KUKA KRL program: EPS_2_26115_SA7010_A_20260219035550.src

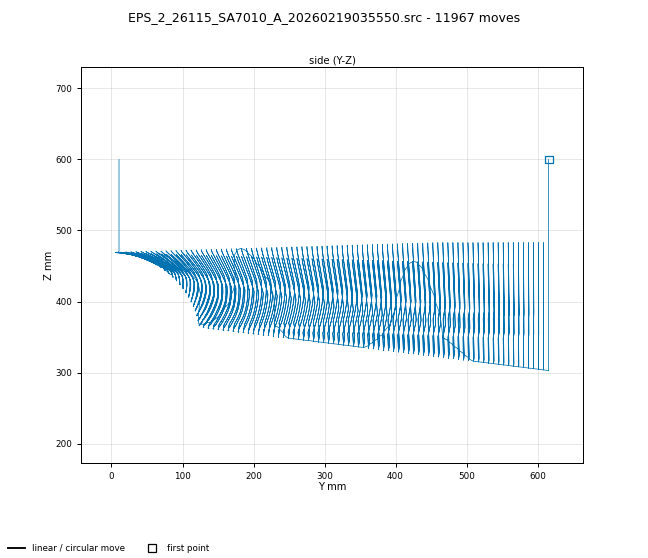
[picture p0: tool path of EPS_2_26115_SA7010_A_20260219035550.src, 11967 of 11969 moves have a stored position in this frame; points joined in program order, loops and branches not executed]
&ACCESS RVP
&REL 4
&COMMENT QRS 19112012
&PARAM EDITMASK = *
DEF PART()
EXT BAS (BAS_COMMAND :IN,REAL :IN )
INT I
BAS (#INITMOV,0 )

;KUKA QRS Post kuka4.cps  Date:22-06-2017 !

File_ID=3066

QRS_PRE_INIT()

;Init var - Until changes are made in qrs_pre_init
Outlet_Square_prg=0
Inlet_1_Square_prg=0
Inlet_2_Square_prg=0
Inlet_3_Square_prg=0
Inlet_4_Square_prg=0
Inlet_5_Square_prg=0

Outlet_1={X 0.000, Y 460.000, Z 382.500, B 0.000, E1 0.000 }
Inlet_1={X 0.000, Y 528.540, Z 352.500, B 0.000, E1 180.000 }
Outlet_1_type=201
Inlet_1_type=201
;QRS#1=Sidecore dimensions
;QRS#2=200-8" PVC SDR 35 Cut Back
;QRS#3=200-8" PVC SDR 35
;QRS#4=
;QRS#5=
;QRS#6=
;QRS#7=
;QRS#8=
;QRS#9=12-08 PSX
;QRS#10=12-08 PSX
;QRS#11=
;QRS#12=
;QRS#13=
;QRS#14=
;QRS#15=
;QRS#16=1220x127x762 2,5'
;QRS#17=EPS Height
;QRS#18=483
;QRS#19=*
;QRS#20= UPDATED VERSION 22-06-2017
;QRS#21=*
Outlet_Square=0100
Inlet_1_Square=0100
Inlet_2_Square=0
Inlet_3_Square=0
Inlet_4_Square=0
Inlet_5_Square=0
Mill_Square=1
Outlet_Square_Prg=214
Inlet_1_Square_prg=204

QRS_INIT()

$ADVANCE=5

; T1
PTP {E1 173.6,E2 173.6}
PTP {X 0,Y 615.497,A -85,B 0,C 180,E1 173.6,E2 173.6,E3 0,E4 0,E5 0,E6 0}
QRS_SPEED_INIT()
LIN {X 0,Y 615.497,Z 600,A -85,B 0,C 180,E1 173.6,E2 173.6,E3 0,E4 0,E5 0,E6 0} C_VEL
LIN {X 0,Y 615.497,Z 312.87,A -85,B 0,C 180,E1 173.6,E2 173.6} C_VEL
LIN {X 0,Y 615.497,Z 304.696,A -85,B 0,C 180,E1 173.6,E2 173.6} C_VEL
LIN {X 0,Y 615.482,Z 302.696,A -85,B 0,C 180,E1 173.414,E2 173.414} C_VEL
LIN {X 0,Y 615.466,Z 302.693,A -85,B 0,C 180,E1 170.801,E2 170.801} C_VEL
LIN {X 0,Y 615.495,Z 302.697,A -85,B 0,C 180,E1 168.139,E2 168.139} C_VEL
LIN {X 0,Y 615.432,Z 302.7,A -85,B 0,C 180,E1 165.449,E2 165.449} C_VEL
LIN {X 0,Y 615.494,Z 302.697,A -85,B 0,C 180,E1 162.73,E2 162.73} C_VEL
LIN {X 0,Y 615.477,Z 302.692,A -85,B 0,C 180,E1 159.967,E2 159.967} C_VEL
LIN {X 0,Y 615.485,Z 302.701,A -85,B 0,C 180,E1 157.651,E2 157.651} C_VEL
LIN {X 0,Y 615.459,Z 302.694,A -85,B 0,C 180,E1 155.007,E2 155.007} C_VEL
LIN {X 0,Y 615.442,Z 302.7,A -85,B 0,C 180,E1 152.083,E2 152.083} C_VEL
LIN {X 0,Y 615.447,Z 302.697,A -85,B 0,C 180,E1 149.838,E2 149.838} C_VEL
LIN {X 0,Y 615.483,Z 302.701,A -85,B 0,C 180,E1 147.542,E2 147.542} C_VEL
LIN {X 0,Y 615.48,Z 302.691,A -85,B 0,C 180,E1 145.184,E2 145.184} C_VEL
LIN {X 0,Y 615.496,Z 302.689,A -85,B 0,C 180,E1 142.758,E2 142.758} C_VEL
LIN {X 0,Y 615.459,Z 302.7,A -85,B 0,C 180,E1 140.247,E2 140.247} C_VEL
LIN {X 0,Y 615.445,Z 302.7,A -85,B 0,C 180,E1 137.643,E2 137.643} C_VEL
LIN {X 0,Y 615.493,Z 302.689,A -85,B 0,C 180,E1 134.932,E2 134.932} C_VEL
LIN {X 0,Y 615.49,Z 302.7,A -85,B 0,C 180,E1 132.08,E2 132.08} C_VEL
LIN {X 0,Y 615.467,Z 302.694,A -85,B 0,C 180,E1 129.75,E2 129.75} C_VEL
LIN {X 0,Y 615.488,Z 302.701,A -85,B 0,C 180,E1 126.936,E2 126.936} C_VEL
LIN {X 0,Y 615.45,Z 302.699,A -85,B 0,C 180,E1 125.617,E2 125.617} C_VEL
LIN {X 0,Y 615.462,Z 303.818,A -85,B 0,C 180,E1 124.697,E2 124.697} C_VEL
LIN {X 0,Y 615.487,Z 307.934,A -85,B 0,C 180,E1 122.33,E2 122.33} C_VEL
LIN {X 0,Y 615.49,Z 313.146,A -85,B 0,C 180,E1 119.405,E2 119.405} C_VEL
LIN {X 0,Y 615.471,Z 317.529,A -85,B 0,C 180,E1 117.041,E2 117.041} C_VEL
LIN {X 0,Y 615.49,Z 322.77,A -85,B 0,C 180,E1 114.271,E2 114.271} C_VEL
LIN {X 0,Y 615.493,Z 328.266,A -85,B 0,C 180,E1 111.431,E2 111.431} C_VEL
LIN {X 0,Y 615.481,Z 333.845,A -85,B 0,C 180,E1 108.602,E2 108.602} C_VEL
LIN {X 0,Y 615.476,Z 339.254,A -85,B 0,C 180,E1 105.905,E2 105.905} C_VEL
LIN {X 0,Y 615.496,Z 344.741,A -85,B 0,C 180,E1 103.2,E2 103.2} C_VEL
LIN {X 0,Y 615.497,Z 348.09,A -85,B 0,C 180,E1 101.568,E2 101.568} C_VEL
LIN {X 0,Y 615.48,Z 362.76,A -85,B 0,C 180,E1 101.234,E2 101.234} C_VEL
LIN {X 0,Y 615.446,Z 375.104,A -85,B 0,C 180,E1 100.825,E2 100.825} C_VEL
LIN {X 0,Y 615.449,Z 387.212,A -85,B 0,C 180,E1 100.278,E2 100.278} C_VEL
LIN {X 0,Y 615.496,Z 398.583,A -85,B 0,C 180,E1 99.613,E2 99.613} C_VEL
LIN {X 0,Y 615.498,Z 408.828,A -85,B 0,C 180,E1 98.867,E2 98.867} C_VEL
LIN {X 0,Y 615.498,Z 418.038,A -85,B 0,C 180,E1 98.04,E2 98.04} C_VEL
LIN {X 0,Y 615.499,Z 426.895,A -85,B 0,C 180,E1 97.057,E2 97.057} C_VEL
LIN {X 0,Y 615.497,Z 434.126,A -85,B 0,C 180,E1 96.062,E2 96.062} C_VEL
LIN {X 0,Y 615.497,Z 438.96,A -85,B 0,C 180,E1 95.241,E2 95.241} C_VEL
LIN {X 0,Y 615.494,Z 443.659,A -85,B 0,C 180,E1 94.256,E2 94.256} C_VEL
LIN {X 0,Y 615.494,Z 447.256,A -85,B 0,C 180,E1 93.273,E2 93.273} C_VEL
LIN {X 0,Y 615.496,Z 449.116,A -85,B 0,C 180,E1 92.617,E2 92.617} C_VEL
LIN {X 0,Y 615.5,Z 450.533,A -85,B 0,C 180,E1 91.963,E2 91.963} C_VEL
LIN {X 0,Y 615.496,Z 452.142,A -85,B 0,C 180,E1 90.654,E2 90.654} C_VEL
LIN {X 0,Y 615.495,Z 452.384,A -85,B 0,C 180,E1 90,E2 90} C_VEL
LIN {X 0,Y 615.495,Z 452.205,A -85,B 0,C 180,E1 89.345,E2 89.345} C_VEL
LIN {X 0,Y 615.5,Z 450.682,A -85,B 0,C 180,E1 88.037,E2 88.037} C_VEL
LIN {X 0,Y 615.498,Z 449.341,A -85,B 0,C 180,E1 87.382,E2 87.382} C_VEL
LIN {X 0,Y 615.496,Z 446.493,A -85,B 0,C 180,E1 86.399,E2 86.399} C_VEL
LIN {X 0,Y 615.498,Z 442.633,A -85,B 0,C 180,E1 85.415,E2 85.415} C_VEL
LIN {X 0,Y 615.498,Z 437.65,A -85,B 0,C 180,E1 84.43,E2 84.43} C_VEL
LIN {X 0,Y 615.496,Z 431.208,A -85,B 0,C 180,E1 83.418,E2 83.418} C_VEL
LIN {X 0,Y 615.497,Z 423.535,A -85,B 0,C 180,E1 82.454,E2 82.454} C_VEL
LIN {X 0,Y 615.498,Z 413.757,A -85,B 0,C 180,E1 81.463,E2 81.463} C_VEL
LIN {X 0,Y 615.498,Z 403.491,A -85,B 0,C 180,E1 80.636,E2 80.636} C_VEL
LIN {X 0,Y 615.459,Z 391.933,A -85,B 0,C 180,E1 79.888,E2 79.888} C_VEL
LIN {X 0,Y 615.436,Z 380.369,A -85,B 0,C 180,E1 79.304,E2 79.304} C_VEL
LIN {X 0,Y 615.462,Z 368.441,A -85,B 0,C 180,E1 78.848,E2 78.848} C_VEL
LIN {X 0,Y 615.491,Z 356.38,A -85,B 0,C 180,E1 78.515,E2 78.515} C_VEL
LIN {X 0,Y 615.497,Z 348.102,A -85,B 0,C 180,E1 78.348,E2 78.348} C_VEL
LIN {X 0,Y 615.474,Z 343.454,A -85,B 0,C 180,E1 76.074,E2 76.074} C_VEL
LIN {X 0,Y 615.463,Z 338.059,A -85,B 0,C 180,E1 73.413,E2 73.413} C_VEL
LIN {X 0,Y 615.49,Z 332.571,A -85,B 0,C 180,E1 70.662,E2 70.662} C_VEL
LIN {X 0,Y 615.473,Z 327.065,A -85,B 0,C 180,E1 67.863,E2 67.863} C_VEL
LIN {X 0,Y 615.488,Z 322.94,A -85,B 0,C 180,E1 65.728,E2 65.728} C_VEL
LIN {X 0,Y 615.474,Z 317.697,A -85,B 0,C 180,E1 62.958,E2 62.958} C_VEL
LIN {X 0,Y 615.492,Z 312.599,A -85,B 0,C 180,E1 60.205,E2 60.205} C_VEL
LIN {X 0,Y 615.488,Z 307.869,A -85,B 0,C 180,E1 57.543,E2 57.543} C_VEL
LIN {X 0,Y 615.467,Z 303.766,A -85,B 0,C 180,E1 55.184,E2 55.184} C_VEL
LIN {X 0,Y 615.454,Z 302.7,A -85,B 0,C 180,E1 54.382,E2 54.382} C_VEL
LIN {X 0,Y 615.449,Z 302.698,A -85,B 0,C 180,E1 51.929,E2 51.929} C_VEL
LIN {X 0,Y 615.49,Z 302.695,A -85,B 0,C 180,E1 49.394,E2 49.394} C_VEL
LIN {X 0,Y 615.489,Z 302.689,A -85,B 0,C 180,E1 46.756,E2 46.756} C_VEL
LIN {X 0,Y 615.458,Z 302.697,A -85,B 0,C 180,E1 43.995,E2 43.995} C_VEL
LIN {X 0,Y 615.481,Z 302.703,A -85,B 0,C 180,E1 41.095,E2 41.095} C_VEL
LIN {X 0,Y 615.474,Z 302.694,A -85,B 0,C 180,E1 38.906,E2 38.906} C_VEL
LIN {X 0,Y 615.464,Z 302.695,A -85,B 0,C 180,E1 36.427,E2 36.427} C_VEL
LIN {X 0,Y 615.483,Z 302.689,A -85,B 0,C 180,E1 33.535,E2 33.535} C_VEL
LIN {X 0,Y 615.495,Z 302.697,A -85,B 0,C 180,E1 30.919,E2 30.919} C_VEL
LIN {X 0,Y 615.439,Z 302.699,A -85,B 0,C 180,E1 28.443,E2 28.443} C_VEL
LIN {X 0,Y 615.498,Z 302.698,A -85,B 0,C 180,E1 25.572,E2 25.572} C_VEL
LIN {X 0,Y 615.463,Z 302.694,A -85,B 0,C 180,E1 22.846,E2 22.846} C_VEL
LIN {X 0,Y 615.491,Z 302.7,A -85,B 0,C 180,E1 20.56,E2 20.56} C_VEL
LIN {X 0,Y 615.473,Z 302.691,A -85,B 0,C 180,E1 17.957,E2 17.957} C_VEL
LIN {X 0,Y 615.478,Z 302.7,A -85,B 0,C 180,E1 15.226,E2 15.226} C_VEL
LIN {X 0,Y 615.439,Z 302.7,A -85,B 0,C 180,E1 12.531,E2 12.531} C_VEL
LIN {X 0,Y 615.497,Z 302.69,A -85,B 0,C 180,E1 9.862,E2 9.862} C_VEL
LIN {X 0,Y 615.476,Z 302.694,A -85,B 0,C 180,E1 7.216,E2 7.216} C_VEL
LIN {X 0,Y 615.468,Z 302.694,A -85,B 0,C 180,E1 4.585,E2 4.585} C_VEL
LIN {X 0,Y 615.499,Z 302.691,A -85,B 0,C 180,E1 1.963,E2 1.963} C_VEL
LIN {X 0,Y 615.438,Z 302.7,A -85,B 0,C 180,E1 -0.654,E2 -0.654} C_VEL
LIN {X 0,Y 615.447,Z 302.696,A -85,B 0,C 180,E1 -2.618,E2 -2.618} C_VEL
LIN {X 0,Y 615.492,Z 302.7,A -85,B 0,C 180,E1 -5.241,E2 -5.241} C_VEL
LIN {X 0,Y 615.488,Z 302.688,A -85,B 0,C 180,E1 -7.876,E2 -7.876} C_VEL
LIN {X 0,Y 615.477,Z 302.699,A -85,B 0,C 180,E1 -10.527,E2 -10.527} C_VEL
LIN {X 0,Y 615.446,Z 302.699,A -85,B 0,C 180,E1 -12.531,E2 -12.531} C_VEL
LIN {X 0,Y 615.469,Z 302.7,A -85,B 0,C 180,E1 -15.227,E2 -15.227} C_VEL
LIN {X 0,Y 615.47,Z 302.692,A -85,B 0,C 180,E1 -17.958,E2 -17.958} C_VEL
LIN {X 0,Y 615.486,Z 302.699,A -85,B 0,C 180,E1 -20.731,E2 -20.731} C_VEL
LIN {X 0,Y 615.489,Z 302.69,A -85,B 0,C 180,E1 -23.556,E2 -23.556} C_VEL
LIN {X 0,Y 615.499,Z 302.7,A -85,B 0,C 180,E1 -25.715,E2 -25.715} C_VEL
LIN {X 0,Y 615.434,Z 302.7,A -85,B 0,C 180,E1 -28.442,E2 -28.442} C_VEL
LIN {X 0,Y 615.495,Z 302.694,A -85,B 0,C 180,E1 -31.088,E2 -31.088} C_VEL
LIN {X 0,Y 615.481,Z 302.696,A -85,B 0,C 180,E1 -34.023,E2 -34.023} C_VEL
LIN {X 0,Y 615.48,Z 302.689,A -85,B 0,C 180,E1 -36.937,E2 -36.937} C_VEL
LIN {X 0,Y 615.46,Z 302.7,A -85,B 0,C 180,E1 -39.752,E2 -39.752} C_VEL
LIN {X 0,Y 615.444,Z 302.7,A -85,B 0,C 180,E1 -42.357,E2 -42.357} C_VEL
LIN {X 0,Y 615.493,Z 302.689,A -85,B 0,C 180,E1 -45.068,E2 -45.068} C_VEL
LIN {X 0,Y 615.49,Z 302.7,A -85,B 0,C 180,E1 -47.92,E2 -47.92} C_VEL
LIN {X 0,Y 615.468,Z 302.694,A -85,B 0,C 180,E1 -50.249,E2 -50.249} C_VEL
LIN {X 0,Y 615.489,Z 302.7,A -85,B 0,C 180,E1 -53.064,E2 -53.064} C_VEL
LIN {X 0,Y 615.468,Z 302.793,A -85,B 0,C 180,E1 -54.584,E2 -54.584} C_VEL
LIN {X 0,Y 615.448,Z 310.011,A -85,B 0,C 180,E1 -57.152,E2 -57.152} C_VEL
LIN {X 0,Y 615.448,Z 317.785,A -85,B 0,C 180,E1 -59.838,E2 -59.838} C_VEL
LIN {X 0,Y 615.496,Z 325.542,A -85,B 0,C 180,E1 -62.455,E2 -62.455} C_VEL
LIN {X 0,Y 615.467,Z 333.312,A -85,B 0,C 180,E1 -65.008,E2 -65.008} C_VEL
LIN {X 0,Y 615.491,Z 341.513,A -85,B 0,C 180,E1 -67.654,E2 -67.654} C_VEL
LIN {X 0,Y 615.484,Z 349.929,A -85,B 0,C 180,E1 -70.315,E2 -70.315} C_VEL
LIN {X 0,Y 615.491,Z 358.782,A -85,B 0,C 180,E1 -73.072,E2 -73.072} C_VEL
LIN {X 0,Y 615.46,Z 367.555,A -85,B 0,C 180,E1 -75.761,E2 -75.761} C_VEL
LIN {X 0,Y 615.497,Z 376.136,A -85,B 0,C 180,E1 -78.369,E2 -78.369} C_VEL
LIN {X 0,Y 615.497,Z 389.818,A -85,B 0,C 180,E1 -78.64,E2 -78.64} C_VEL
LIN {X 0,Y 615.453,Z 402.97,A -85,B 0,C 180,E1 -79.051,E2 -79.051} C_VEL
LIN {X 0,Y 615.442,Z 414.772,A -85,B 0,C 180,E1 -79.555,E2 -79.555} C_VEL
LIN {X 0,Y 615.489,Z 425.386,A -85,B 0,C 180,E1 -80.138,E2 -80.138} C_VEL
LIN {X 0,Y 615.498,Z 436.23,A -85,B 0,C 180,E1 -80.884,E2 -80.884} C_VEL
LIN {X 0,Y 615.497,Z 446.81,A -85,B 0,C 180,E1 -81.794,E2 -81.794} C_VEL
LIN {X 0,Y 615.498,Z 454.605,A -85,B 0,C 180,E1 -82.619,E2 -82.619} C_VEL
LIN {X 0,Y 615.496,Z 462.202,A -85,B 0,C 180,E1 -83.608,E2 -83.608} C_VEL
LIN {X 0,Y 615.498,Z 469.203,A -85,B 0,C 180,E1 -84.759,E2 -84.759} C_VEL
LIN {X 0,Y 615.494,Z 473.85,A -85,B 0,C 180,E1 -85.743,E2 -85.743} C_VEL
LIN {X 0,Y 615.494,Z 477.398,A -85,B 0,C 180,E1 -86.727,E2 -86.727} C_VEL
LIN {X 0,Y 615.497,Z 479.232,A -85,B 0,C 180,E1 -87.382,E2 -87.382} C_VEL
LIN {X 0,Y 615.5,Z 480.607,A -85,B 0,C 180,E1 -88.037,E2 -88.037} C_VEL
LIN {X 0,Y 615.496,Z 482.173,A -85,B 0,C 180,E1 -89.345,E2 -89.345} C_VEL
LIN {X 0,Y 615.494,Z 482.389,A -85,B 0,C 180,E1 -90,E2 -90} C_VEL
LIN {X 0,Y 615.495,Z 481.58,A -85,B 0,C 180,E1 -91.308,E2 -91.308} C_VEL
LIN {X 0,Y 615.5,Z 480.608,A -85,B 0,C 180,E1 -91.963,E2 -91.963} C_VEL
LIN {X 0,Y 615.497,Z 479.234,A -85,B 0,C 180,E1 -92.617,E2 -92.617} C_VEL
LIN {X 0,Y 615.496,Z 476.351,A -85,B 0,C 180,E1 -93.6,E2 -93.6} C_VEL
LIN {X 0,Y 615.498,Z 472.443,A -85,B 0,C 180,E1 -94.584,E2 -94.584} C_VEL
LIN {X 0,Y 615.499,Z 467.407,A -85,B 0,C 180,E1 -95.569,E2 -95.569} C_VEL
LIN {X 0,Y 615.497,Z 460.869,A -85,B 0,C 180,E1 -96.583,E2 -96.583} C_VEL
LIN {X 0,Y 615.497,Z 453.137,A -85,B 0,C 180,E1 -97.545,E2 -97.545} C_VEL
LIN {X 0,Y 615.498,Z 445.05,A -85,B 0,C 180,E1 -98.371,E2 -98.371} C_VEL
LIN {X 0,Y 615.499,Z 435.174,A -85,B 0,C 180,E1 -99.198,E2 -99.198} C_VEL
LIN {X 0,Y 615.479,Z 423.991,A -85,B 0,C 180,E1 -99.945,E2 -99.945} C_VEL
LIN {X 0,Y 615.441,Z 413.04,A -85,B 0,C 180,E1 -100.527,E2 -100.527} C_VEL
LIN {X 0,Y 615.459,Z 400.783,A -85,B 0,C 180,E1 -101.03,E2 -101.03} C_VEL
LIN {X 0,Y 615.499,Z 388.085,A -85,B 0,C 180,E1 -101.401,E2 -101.401} C_VEL
LIN {X 0,Y 615.497,Z 376.138,A -85,B 0,C 180,E1 -101.63,E2 -101.63} C_VEL
LIN {X 0,Y 615.46,Z 367.556,A -85,B 0,C 180,E1 -104.238,E2 -104.238} C_VEL
LIN {X 0,Y 615.491,Z 358.784,A -85,B 0,C 180,E1 -106.928,E2 -106.928} C_VEL
LIN {X 0,Y 615.487,Z 349.931,A -85,B 0,C 180,E1 -109.684,E2 -109.684} C_VEL
LIN {X 0,Y 615.491,Z 341.513,A -85,B 0,C 180,E1 -112.346,E2 -112.346} C_VEL
LIN {X 0,Y 615.467,Z 333.314,A -85,B 0,C 180,E1 -114.992,E2 -114.992} C_VEL
LIN {X 0,Y 615.496,Z 325.544,A -85,B 0,C 180,E1 -117.544,E2 -117.544} C_VEL
LIN {X 0,Y 615.448,Z 317.787,A -85,B 0,C 180,E1 -120.161,E2 -120.161} C_VEL
LIN {X 0,Y 615.448,Z 310.012,A -85,B 0,C 180,E1 -122.847,E2 -122.847} C_VEL
LIN {X 0,Y 615.466,Z 302.699,A -85,B 0,C 180,E1 -125.465,E2 -125.465} C_VEL
LIN {X 0,Y 615.456,Z 302.697,A -85,B 0,C 180,E1 -128.07,E2 -128.07} C_VEL
LIN {X 0,Y 615.486,Z 302.694,A -85,B 0,C 180,E1 -130.605,E2 -130.605} C_VEL
LIN {X 0,Y 615.491,Z 302.69,A -85,B 0,C 180,E1 -133.243,E2 -133.243} C_VEL
LIN {X 0,Y 615.45,Z 302.698,A -85,B 0,C 180,E1 -136.005,E2 -136.005} C_VEL
LIN {X 0,Y 615.456,Z 302.7,A -85,B 0,C 180,E1 -138.523,E2 -138.523} C_VEL
LIN {X 0,Y 615.475,Z 302.693,A -85,B 0,C 180,E1 -141.095,E2 -141.095} C_VEL
LIN {X 0,Y 615.47,Z 302.695,A -85,B 0,C 180,E1 -143.574,E2 -143.574} C_VEL
LIN {X 0,Y 615.481,Z 302.689,A -85,B 0,C 180,E1 -146.465,E2 -146.465} C_VEL
LIN {X 0,Y 615.498,Z 302.698,A -85,B 0,C 180,E1 -149.081,E2 -149.081} C_VEL
LIN {X 0,Y 615.433,Z 302.7,A -85,B 0,C 180,E1 -151.556,E2 -151.556} C_VEL
LIN {X 0,Y 615.494,Z 302.697,A -85,B 0,C 180,E1 -154.427,E2 -154.427} C_VEL
LIN {X 0,Y 615.467,Z 302.694,A -85,B 0,C 180,E1 -157.155,E2 -157.155} C_VEL
LIN {X 0,Y 615.488,Z 302.703,A -85,B 0,C 180,E1 -159.439,E2 -159.439} C_VEL
LIN {X 0,Y 615.469,Z 302.692,A -85,B 0,C 180,E1 -162.042,E2 -162.042} C_VEL
LIN {X 0,Y 615.472,Z 302.7,A -85,B 0,C 180,E1 -164.774,E2 -164.774} C_VEL
LIN {X 0,Y 615.441,Z 302.7,A -85,B 0,C 180,E1 -167.469,E2 -167.469} C_VEL
LIN {X 0,Y 615.497,Z 302.689,A -85,B 0,C 180,E1 -170.138,E2 -170.138} C_VEL
LIN {X 0,Y 615.48,Z 302.694,A -85,B 0,C 180,E1 -172.784,E2 -172.784} C_VEL
LIN {X 0,Y 615.465,Z 302.694,A -85,B 0,C 180,E1 -175.415,E2 -175.415} C_VEL
LIN {X 0,Y 615.499,Z 302.693,A -85,B 0,C 180,E1 -178.037,E2 -178.037} C_VEL
LIN {X 0,Y 615.436,Z 302.7,A -85,B 0,C 180,E1 -180.654,E2 -180.654} C_VEL
LIN {X 0,Y 615.45,Z 302.696,A -85,B 0,C 180,E1 -182.618,E2 -182.618} C_VEL
LIN {X 0,Y 615.49,Z 302.699,A -85,B 0,C 180,E1 -185.241,E2 -185.241} C_VEL
LIN {X 0,Y 615.482,Z 302.696,A -85,B 0,C 180,E1 -186.586,E2 -186.586} C_VEL
LIN {X 0,Y 614.802,Z 302.843,A -85,B 0,C 180,E1 -187.132,E2 -187.132} C_VEL
LIN {X 0,Y 611.956,Z 303.255,A -85,B 0,C 180,E1 -188.018,E2 -188.018} C_VEL
LIN {X 0,Y 609.562,Z 303.564,A -85,B 0,C 180,E1 -188.73,E2 -188.73} C_VEL
LIN {X 0,Y 608.533,Z 303.681,A -85,B 0,C 180,E1 -189.28,E2 -189.28} C_VEL
LIN {X 0,Y 608.449,Z 303.691,A -85,B 0,C 180,E1 -189.466,E2 -189.466} C_VEL
LIN {X 0,Y 608.458,Z 303.698,A -85,B 0,C 180,E1 -192,E2 -192} C_VEL
LIN {X 0,Y 608.405,Z 303.696,A -85,B 0,C 180,E1 -194.722,E2 -194.722} C_VEL
LIN {X 0,Y 608.452,Z 303.693,A -85,B 0,C 180,E1 -197.477,E2 -197.477} C_VEL
LIN {X 0,Y 608.459,Z 303.693,A -85,B 0,C 180,E1 -200.274,E2 -200.274} C_VEL
LIN {X 0,Y 608.448,Z 303.696,A -85,B 0,C 180,E1 -202.477,E2 -202.477} C_VEL
LIN {X 0,Y 608.434,Z 303.693,A -85,B 0,C 180,E1 -204.572,E2 -204.572} C_VEL
LIN {X 0,Y 608.461,Z 303.694,A -85,B 0,C 180,E1 -207.207,E2 -207.207} C_VEL
LIN {X 0,Y 608.42,Z 303.694,A -85,B 0,C 180,E1 -209.966,E2 -209.966} C_VEL
LIN {X 0,Y 608.457,Z 303.697,A -85,B 0,C 180,E1 -212.524,E2 -212.524} C_VEL
LIN {X 0,Y 608.439,Z 303.692,A -85,B 0,C 180,E1 -215.278,E2 -215.278} C_VEL
LIN {X 0,Y 608.46,Z 303.697,A -85,B 0,C 180,E1 -217.747,E2 -217.747} C_VEL
LIN {X 0,Y 608.425,Z 303.694,A -85,B 0,C 180,E1 -220.328,E2 -220.328} C_VEL
LIN {X 0,Y 608.463,Z 303.69,A -85,B 0,C 180,E1 -223.31,E2 -223.31} C_VEL
LIN {X 0,Y 608.462,Z 303.695,A -85,B 0,C 180,E1 -226.131,E2 -226.131} C_VEL
LIN {X 0,Y 608.455,Z 303.69,A -85,B 0,C 180,E1 -228.825,E2 -228.825} C_VEL
LIN {X 0,Y 608.463,Z 303.697,A -85,B 0,C 180,E1 -231.413,E2 -231.413} C_VEL
LIN {X 0,Y 608.427,Z 303.693,A -85,B 0,C 180,E1 -233.957,E2 -233.957} C_VEL
LIN {X 0,Y 608.389,Z 303.802,A -85,B 0,C 180,E1 -234.72,E2 -234.72} C_VEL
LIN {X 0,Y 608.462,Z 307.941,A -85,B 0,C 180,E1 -237.122,E2 -237.122} C_VEL
LIN {X 0,Y 608.452,Z 313.03,A -85,B 0,C 180,E1 -240.031,E2 -240.031} C_VEL
LIN {X 0,Y 608.43,Z 318.103,A -85,B 0,C 180,E1 -242.802,E2 -242.802} C_VEL
LIN {X 0,Y 608.421,Z 323.038,A -85,B 0,C 180,E1 -245.428,E2 -245.428} C_VEL
LIN {X 0,Y 608.446,Z 328.567,A -85,B 0,C 180,E1 -248.308,E2 -248.308} C_VEL
LIN {X 0,Y 608.422,Z 334.429,A -85,B 0,C 180,E1 -251.298,E2 -251.298} C_VEL
LIN {X 0,Y 608.431,Z 339.626,A -85,B 0,C 180,E1 -253.906,E2 -253.906} C_VEL
LIN {X 0,Y 608.435,Z 345.156,A -85,B 0,C 180,E1 -256.643,E2 -256.643} C_VEL
LIN {X 0,Y 608.449,Z 348.525,A -85,B 0,C 180,E1 -258.296,E2 -258.296} C_VEL
LIN {X 0,Y 608.529,Z 364.411,A -85,B 0,C 180,E1 -258.678,E2 -258.678} C_VEL
LIN {X 0,Y 608.478,Z 376.8,A -85,B 0,C 180,E1 -259.112,E2 -259.112} C_VEL
LIN {X 0,Y 608.454,Z 388.944,A -85,B 0,C 180,E1 -259.687,E2 -259.687} C_VEL
LIN {X 0,Y 608.497,Z 400.074,A -85,B 0,C 180,E1 -260.36,E2 -260.36} C_VEL
LIN {X 0,Y 608.474,Z 409.09,A -85,B 0,C 180,E1 -261.03,E2 -261.03} C_VEL
LIN {X 0,Y 608.464,Z 418.354,A -85,B 0,C 180,E1 -261.866,E2 -261.866} C_VEL
LIN {X 0,Y 608.466,Z 427.327,A -85,B 0,C 180,E1 -262.868,E2 -262.868} C_VEL
LIN {X 0,Y 608.444,Z 434.558,A -85,B 0,C 180,E1 -263.867,E2 -263.867} C_VEL
LIN {X 0,Y 608.462,Z 439.436,A -85,B 0,C 180,E1 -264.699,E2 -264.699} C_VEL
LIN {X 0,Y 608.439,Z 444.18,A -85,B 0,C 180,E1 -265.695,E2 -265.695} C_VEL
LIN {X 0,Y 608.425,Z 447.813,A -85,B 0,C 180,E1 -266.689,E2 -266.689} C_VEL
LIN {X 0,Y 608.425,Z 449.692,A -85,B 0,C 180,E1 -267.352,E2 -267.352} C_VEL
LIN {X 0,Y 608.445,Z 451.127,A -85,B 0,C 180,E1 -268.015,E2 -268.015} C_VEL
LIN {X 0,Y 608.439,Z 452.752,A -85,B 0,C 180,E1 -269.338,E2 -269.338} C_VEL
LIN {X 0,Y 608.435,Z 452.995,A -85,B 0,C 180,E1 -270,E2 -270} C_VEL
LIN {X 0,Y 608.438,Z 452.815,A -85,B 0,C 180,E1 -270.662,E2 -270.662} C_VEL
LIN {X 0,Y 608.445,Z 451.276,A -85,B 0,C 180,E1 -271.986,E2 -271.986} C_VEL
LIN {X 0,Y 608.426,Z 449.918,A -85,B 0,C 180,E1 -272.649,E2 -272.649} C_VEL
LIN {X 0,Y 608.449,Z 447.041,A -85,B 0,C 180,E1 -273.643,E2 -273.643} C_VEL
LIN {X 0,Y 608.433,Z 443.142,A -85,B 0,C 180,E1 -274.638,E2 -274.638} C_VEL
LIN {X 0,Y 608.45,Z 438.111,A -85,B 0,C 180,E1 -275.635,E2 -275.635} C_VEL
LIN {X 0,Y 608.441,Z 431.794,A -85,B 0,C 180,E1 -276.633,E2 -276.633} C_VEL
LIN {X 0,Y 608.475,Z 423.877,A -85,B 0,C 180,E1 -277.633,E2 -277.633} C_VEL
LIN {X 0,Y 608.472,Z 414.035,A -85,B 0,C 180,E1 -278.636,E2 -278.636} C_VEL
LIN {X 0,Y 608.481,Z 403.712,A -85,B 0,C 180,E1 -279.473,E2 -279.473} C_VEL
LIN {X 0,Y 608.471,Z 392.098,A -85,B 0,C 180,E1 -280.229,E2 -280.229} C_VEL
LIN {X 0,Y 608.463,Z 380.492,A -85,B 0,C 180,E1 -280.82,E2 -280.82} C_VEL
LIN {X 0,Y 608.492,Z 368.423,A -85,B 0,C 180,E1 -281.286,E2 -281.286} C_VEL
LIN {X 0,Y 608.537,Z 355.557,A -85,B 0,C 180,E1 -281.639,E2 -281.639} C_VEL
LIN {X 0,Y 608.441,Z 348.536,A -85,B 0,C 180,E1 -281.789,E2 -281.789} C_VEL
LIN {X 0,Y 608.427,Z 343.954,A -85,B 0,C 180,E1 -284.038,E2 -284.038} C_VEL
LIN {X 0,Y 608.405,Z 338.422,A -85,B 0,C 180,E1 -286.785,E2 -286.785} C_VEL
LIN {X 0,Y 608.43,Z 332.89,A -85,B 0,C 180,E1 -289.571,E2 -289.571} C_VEL
LIN {X 0,Y 608.435,Z 327.357,A -85,B 0,C 180,E1 -292.407,E2 -292.407} C_VEL
LIN {X 0,Y 608.421,Z 323.208,A -85,B 0,C 180,E1 -294.572,E2 -294.572} C_VEL
LIN {X 0,Y 608.432,Z 318.269,A -85,B 0,C 180,E1 -297.198,E2 -297.198} C_VEL
LIN {X 0,Y 608.453,Z 313.188,A -85,B 0,C 180,E1 -299.969,E2 -299.969} C_VEL
LIN {X 0,Y 608.46,Z 308.059,A -85,B 0,C 180,E1 -302.879,E2 -302.879} C_VEL
LIN {X 0,Y 608.392,Z 303.954,A -85,B 0,C 180,E1 -305.281,E2 -305.281} C_VEL
LIN {X 0,Y 608.479,Z 303.692,A -85,B 0,C 180,E1 -307.159,E2 -307.159} C_VEL
LIN {X 0,Y 608.446,Z 303.698,A -85,B 0,C 180,E1 -310.328,E2 -310.328} C_VEL
LIN {X 0,Y 608.455,Z 303.69,A -85,B 0,C 180,E1 -312.959,E2 -312.959} C_VEL
LIN {X 0,Y 608.441,Z 303.696,A -85,B 0,C 180,E1 -315.737,E2 -315.737} C_VEL
LIN {X 0,Y 608.417,Z 303.695,A -85,B 0,C 180,E1 -317.935,E2 -317.935} C_VEL
LIN {X 0,Y 608.439,Z 303.699,A -85,B 0,C 180,E1 -320.705,E2 -320.705} C_VEL
LIN {X 0,Y 608.448,Z 303.691,A -85,B 0,C 180,E1 -323.084,E2 -323.084} C_VEL
LIN {X 0,Y 608.464,Z 303.693,A -85,B 0,C 180,E1 -325.53,E2 -325.53} C_VEL
LIN {X 0,Y 608.461,Z 303.691,A -85,B 0,C 180,E1 -327.905,E2 -327.905} C_VEL
LIN {X 0,Y 608.445,Z 303.691,A -85,B 0,C 180,E1 -330.219,E2 -330.219} C_VEL
LIN {X 0,Y 608.465,Z 303.694,A -85,B 0,C 180,E1 -332.794,E2 -332.794} C_VEL
LIN {X 0,Y 608.431,Z 303.693,A -85,B 0,C 180,E1 -335.428,E2 -335.428} C_VEL
LIN {X 0,Y 608.473,Z 303.689,A -85,B 0,C 180,E1 -338.308,E2 -338.308} C_VEL
LIN {X 0,Y 608.466,Z 303.695,A -85,B 0,C 180,E1 -341.283,E2 -341.283} C_VEL
LIN {X 0,Y 608.441,Z 303.692,A -85,B 0,C 180,E1 -343.906,E2 -343.906} C_VEL
LIN {X 0,Y 608.433,Z 303.696,A -85,B 0,C 180,E1 -346.643,E2 -346.643} C_VEL
LIN {X 0,Y 608.439,Z 303.694,A -85,B 0,C 180,E1 -349.35,E2 -349.35} C_VEL
LIN {X 0,Y 608.479,Z 303.688,A -85,B 0,C 180,E1 -352.033,E2 -352.033} C_VEL
LIN {X 0,Y 608.468,Z 303.693,A -85,B 0,C 180,E1 -354.698,E2 -354.698} C_VEL
LIN {X 0,Y 608.448,Z 303.691,A -85,B 0,C 180,E1 -357.352,E2 -357.352} C_VEL
LIN {X 0,Y 608.47,Z 303.695,A -85,B 0,C 180,E1 -360,E2 -360} C_VEL
LIN {X 0,Y 608.442,Z 303.691,A -85,B 0,C 180,E1 -362.648,E2 -362.648} C_VEL
LIN {X 0,Y 608.471,Z 303.694,A -85,B 0,C 180,E1 -365.302,E2 -365.302} C_VEL
LIN {X 0,Y 608.479,Z 303.687,A -85,B 0,C 180,E1 -367.967,E2 -367.967} C_VEL
LIN {X 0,Y 608.449,Z 303.691,A -85,B 0,C 180,E1 -370.95,E2 -370.95} C_VEL
LIN {X 0,Y 608.434,Z 303.695,A -85,B 0,C 180,E1 -373.357,E2 -373.357} C_VEL
LIN {X 0,Y 608.437,Z 303.693,A -85,B 0,C 180,E1 -376.094,E2 -376.094} C_VEL
LIN {X 0,Y 608.451,Z 303.698,A -85,B 0,C 180,E1 -378.87,E2 -378.87} C_VEL
LIN {X 0,Y 608.473,Z 303.688,A -85,B 0,C 180,E1 -381.691,E2 -381.691} C_VEL
LIN {X 0,Y 608.437,Z 303.693,A -85,B 0,C 180,E1 -384.572,E2 -384.572} C_VEL
LIN {X 0,Y 608.462,Z 303.693,A -85,B 0,C 180,E1 -387.206,E2 -387.206} C_VEL
LIN {X 0,Y 608.42,Z 303.694,A -85,B 0,C 180,E1 -389.965,E2 -389.965} C_VEL
LIN {X 0,Y 608.458,Z 303.697,A -85,B 0,C 180,E1 -392.523,E2 -392.523} C_VEL
LIN {X 0,Y 608.439,Z 303.692,A -85,B 0,C 180,E1 -395.278,E2 -395.278} C_VEL
LIN {X 0,Y 608.462,Z 303.697,A -85,B 0,C 180,E1 -397.747,E2 -397.747} C_VEL
LIN {X 0,Y 608.429,Z 303.693,A -85,B 0,C 180,E1 -400.327,E2 -400.327} C_VEL
LIN {X 0,Y 608.463,Z 303.691,A -85,B 0,C 180,E1 -403.309,E2 -403.309} C_VEL
LIN {X 0,Y 608.462,Z 303.695,A -85,B 0,C 180,E1 -406.131,E2 -406.131} C_VEL
LIN {X 0,Y 608.455,Z 303.69,A -85,B 0,C 180,E1 -408.824,E2 -408.824} C_VEL
LIN {X 0,Y 608.447,Z 303.694,A -85,B 0,C 180,E1 -411.762,E2 -411.762} C_VEL
LIN {X 0,Y 608.431,Z 303.696,A -85,B 0,C 180,E1 -414.417,E2 -414.417} C_VEL
LIN {X 0,Y 608.466,Z 311.17,A -85,B 0,C 180,E1 -417.121,E2 -417.121} C_VEL
LIN {X 0,Y 608.473,Z 319.511,A -85,B 0,C 180,E1 -420.028,E2 -420.028} C_VEL
LIN {X 0,Y 608.469,Z 327.684,A -85,B 0,C 180,E1 -422.795,E2 -422.795} C_VEL
LIN {X 0,Y 608.448,Z 335.657,A -85,B 0,C 180,E1 -425.429,E2 -425.429} C_VEL
LIN {X 0,Y 608.478,Z 344.561,A -85,B 0,C 180,E1 -428.309,E2 -428.309} C_VEL
LIN {X 0,Y 608.461,Z 353.466,A -85,B 0,C 180,E1 -431.131,E2 -431.131} C_VEL
LIN {X 0,Y 608.433,Z 362.37,A -85,B 0,C 180,E1 -433.905,E2 -433.905} C_VEL
LIN {X 0,Y 608.443,Z 371.274,A -85,B 0,C 180,E1 -436.643,E2 -436.643} C_VEL
LIN {X 0,Y 608.436,Z 376.491,A -85,B 0,C 180,E1 -438.232,E2 -438.232} C_VEL
LIN {X 0,Y 608.546,Z 390.694,A -85,B 0,C 180,E1 -438.53,E2 -438.53} C_VEL
LIN {X 0,Y 608.496,Z 403.799,A -85,B 0,C 180,E1 -438.951,E2 -438.951} C_VEL
LIN {X 0,Y 608.47,Z 414.919,A -85,B 0,C 180,E1 -439.434,E2 -439.434} C_VEL
LIN {X 0,Y 608.478,Z 425.577,A -85,B 0,C 180,E1 -440.023,E2 -440.023} C_VEL
LIN {X 0,Y 608.483,Z 436.472,A -85,B 0,C 180,E1 -440.778,E2 -440.778} C_VEL
LIN {X 0,Y 608.475,Z 447.11,A -85,B 0,C 180,E1 -441.699,E2 -441.699} C_VEL
LIN {X 0,Y 608.471,Z 454.959,A -85,B 0,C 180,E1 -442.534,E2 -442.534} C_VEL
LIN {X 0,Y 608.461,Z 462.286,A -85,B 0,C 180,E1 -443.484,E2 -443.484} C_VEL
LIN {X 0,Y 608.451,Z 467.865,A -85,B 0,C 180,E1 -444.365,E2 -444.365} C_VEL
LIN {X 0,Y 608.432,Z 472.949,A -85,B 0,C 180,E1 -445.362,E2 -445.362} C_VEL
LIN {X 0,Y 608.449,Z 476.895,A -85,B 0,C 180,E1 -446.357,E2 -446.357} C_VEL
LIN {X 0,Y 608.425,Z 479.808,A -85,B 0,C 180,E1 -447.351,E2 -447.351} C_VEL
LIN {X 0,Y 608.445,Z 481.201,A -85,B 0,C 180,E1 -448.014,E2 -448.014} C_VEL
LIN {X 0,Y 608.438,Z 482.783,A -85,B 0,C 180,E1 -449.338,E2 -449.338} C_VEL
LIN {X 0,Y 608.434,Z 483,A -85,B 0,C 180,E1 -450,E2 -450} C_VEL
LIN {X 0,Y 608.448,Z 482.184,A -85,B 0,C 180,E1 -451.323,E2 -451.323} C_VEL
LIN {X 0,Y 608.445,Z 481.202,A -85,B 0,C 180,E1 -451.985,E2 -451.985} C_VEL
LIN {X 0,Y 608.425,Z 479.81,A -85,B 0,C 180,E1 -452.648,E2 -452.648} C_VEL
LIN {X 0,Y 608.449,Z 476.897,A -85,B 0,C 180,E1 -453.642,E2 -453.642} C_VEL
LIN {X 0,Y 608.432,Z 472.952,A -85,B 0,C 180,E1 -454.637,E2 -454.637} C_VEL
LIN {X 0,Y 608.438,Z 466.879,A -85,B 0,C 180,E1 -455.8,E2 -455.8} C_VEL
LIN {X 0,Y 608.462,Z 460.238,A -85,B 0,C 180,E1 -456.799,E2 -456.799} C_VEL
LIN {X 0,Y 608.456,Z 451.993,A -85,B 0,C 180,E1 -457.8,E2 -457.8} C_VEL
LIN {X 0,Y 608.472,Z 443.541,A -85,B 0,C 180,E1 -458.635,E2 -458.635} C_VEL
LIN {X 0,Y 608.48,Z 433.097,A -85,B 0,C 180,E1 -459.473,E2 -459.473} C_VEL
LIN {X 0,Y 608.488,Z 422.763,A -85,B 0,C 180,E1 -460.144,E2 -460.144} C_VEL
LIN {X 0,Y 608.466,Z 411.861,A -85,B 0,C 180,E1 -460.713,E2 -460.713} C_VEL
LIN {X 0,Y 608.492,Z 400.099,A -85,B 0,C 180,E1 -461.186,E2 -461.186} C_VEL
LIN {X 0,Y 608.55,Z 387.289,A -85,B 0,C 180,E1 -461.554,E2 -461.554} C_VEL
LIN {X 0,Y 608.437,Z 376.493,A -85,B 0,C 180,E1 -461.767,E2 -461.767} C_VEL
LIN {X 0,Y 608.405,Z 367.937,A -85,B 0,C 180,E1 -464.38,E2 -464.38} C_VEL
LIN {X 0,Y 608.45,Z 360.146,A -85,B 0,C 180,E1 -466.783,E2 -466.783} C_VEL
LIN {X 0,Y 608.46,Z 351.241,A -85,B 0,C 180,E1 -469.57,E2 -469.57} C_VEL
LIN {X 0,Y 608.459,Z 342.118,A -85,B 0,C 180,E1 -472.476,E2 -472.476} C_VEL
LIN {X 0,Y 608.453,Z 334.546,A -85,B 0,C 180,E1 -474.935,E2 -474.935} C_VEL
LIN {X 0,Y 608.475,Z 326.755,A -85,B 0,C 180,E1 -477.516,E2 -477.516} C_VEL
LIN {X 0,Y 608.473,Z 319.511,A -85,B 0,C 180,E1 -479.972,E2 -479.972} C_VEL
LIN {X 0,Y 608.466,Z 311.172,A -85,B 0,C 180,E1 -482.878,E2 -482.878} C_VEL
LIN {X 0,Y 608.434,Z 303.696,A -85,B 0,C 180,E1 -485.582,E2 -485.582} C_VEL
LIN {X 0,Y 608.447,Z 303.694,A -85,B 0,C 180,E1 -488.237,E2 -488.237} C_VEL
LIN {X 0,Y 608.449,Z 303.698,A -85,B 0,C 180,E1 -490.328,E2 -490.328} C_VEL
LIN {X 0,Y 608.455,Z 303.69,A -85,B 0,C 180,E1 -492.958,E2 -492.958} C_VEL
LIN {X 0,Y 608.433,Z 303.696,A -85,B 0,C 180,E1 -495.737,E2 -495.737} C_VEL
LIN {X 0,Y 608.416,Z 303.695,A -85,B 0,C 180,E1 -497.935,E2 -497.935} C_VEL
LIN {X 0,Y 608.47,Z 303.694,A -85,B 0,C 180,E1 -500.701,E2 -500.701} C_VEL
LIN {X 0,Y 608.45,Z 303.69,A -85,B 0,C 180,E1 -503.084,E2 -503.084} C_VEL
LIN {X 0,Y 608.464,Z 303.694,A -85,B 0,C 180,E1 -505.53,E2 -505.53} C_VEL
LIN {X 0,Y 608.455,Z 303.691,A -85,B 0,C 180,E1 -507.905,E2 -507.905} C_VEL
LIN {X 0,Y 608.441,Z 303.692,A -85,B 0,C 180,E1 -510.219,E2 -510.219} C_VEL
LIN {X 0,Y 608.461,Z 303.694,A -85,B 0,C 180,E1 -512.793,E2 -512.793} C_VEL
LIN {X 0,Y 608.434,Z 303.693,A -85,B 0,C 180,E1 -515.428,E2 -515.428} C_VEL
LIN {X 0,Y 608.473,Z 303.688,A -85,B 0,C 180,E1 -518.309,E2 -518.309} C_VEL
LIN {X 0,Y 608.46,Z 303.695,A -85,B 0,C 180,E1 -521.283,E2 -521.283} C_VEL
LIN {X 0,Y 608.438,Z 303.692,A -85,B 0,C 180,E1 -523.906,E2 -523.906} C_VEL
LIN {X 0,Y 608.431,Z 303.696,A -85,B 0,C 180,E1 -526.643,E2 -526.643} C_VEL
LIN {X 0,Y 608.444,Z 303.694,A -85,B 0,C 180,E1 -529.35,E2 -529.35} C_VEL
LIN {X 0,Y 608.478,Z 303.688,A -85,B 0,C 180,E1 -532.033,E2 -532.033} C_VEL
LIN {X 0,Y 608.47,Z 303.694,A -85,B 0,C 180,E1 -534.698,E2 -534.698} C_VEL
LIN {X 0,Y 608.444,Z 303.691,A -85,B 0,C 180,E1 -537.352,E2 -537.352} C_VEL
LIN {X 0,Y 608.467,Z 303.697,A -85,B 0,C 180,E1 -540,E2 -540} C_VEL
LIN {X 0,Y 608.444,Z 303.691,A -85,B 0,C 180,E1 -542.648,E2 -542.648} C_VEL
LIN {X 0,Y 608.469,Z 303.694,A -85,B 0,C 180,E1 -545.302,E2 -545.302} C_VEL
LIN {X 0,Y 608.478,Z 303.688,A -85,B 0,C 180,E1 -547.967,E2 -547.967} C_VEL
LIN {X 0,Y 608.449,Z 303.691,A -85,B 0,C 180,E1 -549.466,E2 -549.466} C_VEL
LIN {X 0,Y 607.783,Z 303.779,A -85,B 0,C 180,E1 -550.019,E2 -550.019} C_VEL
LIN {X 0,Y 604.936,Z 304.135,A -85,B 0,C 180,E1 -550.916,E2 -550.916} C_VEL
LIN {X 0,Y 602.523,Z 304.436,A -85,B 0,C 180,E1 -551.637,E2 -551.637} C_VEL
LIN {X 0,Y 601.478,Z 304.564,A -85,B 0,C 180,E1 -552.193,E2 -552.193} C_VEL
LIN {X 0,Y 601.388,Z 304.573,A -85,B 0,C 180,E1 -552.382,E2 -552.382} C_VEL
LIN {X 0,Y 601.381,Z 304.572,A -85,B 0,C 180,E1 -554.898,E2 -554.898} C_VEL
LIN {X 0,Y 601.403,Z 304.574,A -85,B 0,C 180,E1 -556.987,E2 -556.987} C_VEL
LIN {X 0,Y 601.403,Z 304.568,A -85,B 0,C 180,E1 -559.81,E2 -559.81} C_VEL
LIN {X 0,Y 601.405,Z 304.571,A -85,B 0,C 180,E1 -562.606,E2 -562.606} C_VEL
LIN {X 0,Y 601.388,Z 304.57,A -85,B 0,C 180,E1 -564.879,E2 -564.879} C_VEL
LIN {X 0,Y 601.395,Z 304.577,A -85,B 0,C 180,E1 -567.361,E2 -567.361} C_VEL
LIN {X 0,Y 601.391,Z 304.57,A -85,B 0,C 180,E1 -570.166,E2 -570.166} C_VEL
LIN {X 0,Y 601.419,Z 304.572,A -85,B 0,C 180,E1 -572.717,E2 -572.717} C_VEL
LIN {X 0,Y 601.405,Z 304.568,A -85,B 0,C 180,E1 -575.115,E2 -575.115} C_VEL
LIN {X 0,Y 601.43,Z 304.569,A -85,B 0,C 180,E1 -577.42,E2 -577.42} C_VEL
LIN {X 0,Y 601.38,Z 304.572,A -85,B 0,C 180,E1 -579.998,E2 -579.998} C_VEL
LIN {X 0,Y 601.379,Z 304.577,A -85,B 0,C 180,E1 -582.673,E2 -582.673} C_VEL
LIN {X 0,Y 601.421,Z 304.566,A -85,B 0,C 180,E1 -585.483,E2 -585.483} C_VEL
LIN {X 0,Y 601.423,Z 304.568,A -85,B 0,C 180,E1 -588.407,E2 -588.407} C_VEL
LIN {X 0,Y 601.434,Z 304.566,A -85,B 0,C 180,E1 -590.876,E2 -590.876} C_VEL
LIN {X 0,Y 601.397,Z 304.573,A -85,B 0,C 180,E1 -593.418,E2 -593.418} C_VEL
LIN {X 0,Y 601.359,Z 304.575,A -85,B 0,C 180,E1 -594.245,E2 -594.245} C_VEL
LIN {X 0,Y 601.381,Z 305.238,A -85,B 0,C 180,E1 -595.067,E2 -595.067} C_VEL
LIN {X 0,Y 601.434,Z 309.378,A -85,B 0,C 180,E1 -597.486,E2 -597.486} C_VEL
LIN {X 0,Y 601.378,Z 314.773,A -85,B 0,C 180,E1 -600.606,E2 -600.606} C_VEL
LIN {X 0,Y 601.374,Z 318.893,A -85,B 0,C 180,E1 -602.886,E2 -602.886} C_VEL
LIN {X 0,Y 601.38,Z 324.163,A -85,B 0,C 180,E1 -605.72,E2 -605.72} C_VEL
LIN {X 0,Y 601.354,Z 328.568,A -85,B 0,C 180,E1 -608.039,E2 -608.039} C_VEL
LIN {X 0,Y 601.348,Z 334.097,A -85,B 0,C 180,E1 -610.899,E2 -610.899} C_VEL
LIN {X 0,Y 601.339,Z 339.627,A -85,B 0,C 180,E1 -613.711,E2 -613.711} C_VEL
LIN {X 0,Y 601.332,Z 345.157,A -85,B 0,C 180,E1 -616.483,E2 -616.483} C_VEL
LIN {X 0,Y 601.345,Z 348.527,A -85,B 0,C 180,E1 -618.156,E2 -618.156} C_VEL
LIN {X 0,Y 601.603,Z 353.418,A -85,B 0,C 180,E1 -618.268,E2 -618.268} C_VEL
LIN {X 0,Y 601.557,Z 365.756,A -85,B 0,C 180,E1 -618.585,E2 -618.585} C_VEL
LIN {X 0,Y 601.499,Z 378.364,A -85,B 0,C 180,E1 -619.052,E2 -619.052} C_VEL
LIN {X 0,Y 601.455,Z 390.522,A -85,B 0,C 180,E1 -619.651,E2 -619.651} C_VEL
LIN {X 0,Y 601.467,Z 401.317,A -85,B 0,C 180,E1 -620.331,E2 -620.331} C_VEL
LIN {X 0,Y 601.434,Z 411.089,A -85,B 0,C 180,E1 -621.093,E2 -621.093} C_VEL
LIN {X 0,Y 601.407,Z 419.985,A -85,B 0,C 180,E1 -621.939,E2 -621.939} C_VEL
LIN {X 0,Y 601.406,Z 428.67,A -85,B 0,C 180,E1 -622.952,E2 -622.952} C_VEL
LIN {X 0,Y 601.361,Z 435.599,A -85,B 0,C 180,E1 -623.963,E2 -623.963} C_VEL
LIN {X 0,Y 601.344,Z 441.151,A -85,B 0,C 180,E1 -624.972,E2 -624.972} C_VEL
LIN {X 0,Y 601.347,Z 445.512,A -85,B 0,C 180,E1 -625.979,E2 -625.979} C_VEL
LIN {X 0,Y 601.344,Z 447.816,A -85,B 0,C 180,E1 -626.65,E2 -626.65} C_VEL
LIN {X 0,Y 601.324,Z 449.694,A -85,B 0,C 180,E1 -627.321,E2 -627.321} C_VEL
LIN {X 0,Y 601.343,Z 451.128,A -85,B 0,C 180,E1 -627.991,E2 -627.991} C_VEL
LIN {X 0,Y 601.339,Z 452.753,A -85,B 0,C 180,E1 -629.331,E2 -629.331} C_VEL
LIN {X 0,Y 601.336,Z 452.996,A -85,B 0,C 180,E1 -630,E2 -630} C_VEL
LIN {X 0,Y 601.339,Z 452.815,A -85,B 0,C 180,E1 -630.67,E2 -630.67} C_VEL
LIN {X 0,Y 601.344,Z 451.275,A -85,B 0,C 180,E1 -632.01,E2 -632.01} C_VEL
LIN {X 0,Y 601.326,Z 449.916,A -85,B 0,C 180,E1 -632.68,E2 -632.68} C_VEL
LIN {X 0,Y 601.368,Z 447.039,A -85,B 0,C 180,E1 -633.686,E2 -633.686} C_VEL
LIN {X 0,Y 601.337,Z 443.14,A -85,B 0,C 180,E1 -634.693,E2 -634.693} C_VEL
LIN {X 0,Y 601.373,Z 438.108,A -85,B 0,C 180,E1 -635.701,E2 -635.701} C_VEL
LIN {X 0,Y 601.382,Z 431.79,A -85,B 0,C 180,E1 -636.711,E2 -636.711} C_VEL
LIN {X 0,Y 601.396,Z 423.873,A -85,B 0,C 180,E1 -637.724,E2 -637.724} C_VEL
LIN {X 0,Y 601.437,Z 414.029,A -85,B 0,C 180,E1 -638.738,E2 -638.738} C_VEL
LIN {X 0,Y 601.449,Z 403.706,A -85,B 0,C 180,E1 -639.585,E2 -639.585} C_VEL
LIN {X 0,Y 601.45,Z 392.088,A -85,B 0,C 180,E1 -640.35,E2 -640.35} C_VEL
LIN {X 0,Y 601.486,Z 379.979,A -85,B 0,C 180,E1 -640.969,E2 -640.969} C_VEL
LIN {X 0,Y 601.546,Z 367.244,A -85,B 0,C 180,E1 -641.456,E2 -641.456} C_VEL
LIN {X 0,Y 601.609,Z 354.618,A -85,B 0,C 180,E1 -641.796,E2 -641.796} C_VEL
LIN {X 0,Y 601.338,Z 348.534,A -85,B 0,C 180,E1 -641.93,E2 -641.93} C_VEL
LIN {X 0,Y 601.329,Z 342.57,A -85,B 0,C 180,E1 -644.899,E2 -644.899} C_VEL
LIN {X 0,Y 601.329,Z 337.038,A -85,B 0,C 180,E1 -647.69,E2 -647.69} C_VEL
LIN {X 0,Y 601.341,Z 331.506,A -85,B 0,C 180,E1 -650.525,E2 -650.525} C_VEL
LIN {X 0,Y 601.366,Z 325.973,A -85,B 0,C 180,E1 -653.412,E2 -653.412} C_VEL
LIN {X 0,Y 601.355,Z 320.44,A -85,B 0,C 180,E1 -656.366,E2 -656.366} C_VEL
LIN {X 0,Y 601.354,Z 316.035,A -85,B 0,C 180,E1 -658.774,E2 -658.774} C_VEL
LIN {X 0,Y 601.379,Z 311.323,A -85,B 0,C 180,E1 -661.448,E2 -661.448} C_VEL
LIN {X 0,Y 601.427,Z 306.769,A -85,B 0,C 180,E1 -664.118,E2 -664.118} C_VEL
LIN {X 0,Y 601.363,Z 305.099,A -85,B 0,C 180,E1 -665.107,E2 -665.107} C_VEL
LIN {X 0,Y 601.361,Z 304.575,A -85,B 0,C 180,E1 -665.756,E2 -665.756} C_VEL
LIN {X 0,Y 601.395,Z 304.572,A -85,B 0,C 180,E1 -668.269,E2 -668.269} C_VEL
LIN {X 0,Y 601.415,Z 304.568,A -85,B 0,C 180,E1 -670.874,E2 -670.874} C_VEL
LIN {X 0,Y 601.428,Z 304.57,A -85,B 0,C 180,E1 -673.586,E2 -673.586} C_VEL
LIN {X 0,Y 601.404,Z 304.568,A -85,B 0,C 180,E1 -676.429,E2 -676.429} C_VEL
LIN {X 0,Y 601.4,Z 304.57,A -85,B 0,C 180,E1 -679.428,E2 -679.428} C_VEL
LIN {X 0,Y 601.397,Z 304.57,A -85,B 0,C 180,E1 -681.73,E2 -681.73} C_VEL
LIN {X 0,Y 601.404,Z 304.574,A -85,B 0,C 180,E1 -684.246,E2 -684.246} C_VEL
LIN {X 0,Y 601.427,Z 304.565,A -85,B 0,C 180,E1 -686.686,E2 -686.686} C_VEL
LIN {X 0,Y 601.418,Z 304.572,A -85,B 0,C 180,E1 -689.058,E2 -689.058} C_VEL
LIN {X 0,Y 601.399,Z 304.571,A -85,B 0,C 180,E1 -691.371,E2 -691.371} C_VEL
LIN {X 0,Y 601.403,Z 304.573,A -85,B 0,C 180,E1 -694.133,E2 -694.133} C_VEL
LIN {X 0,Y 601.414,Z 304.568,A -85,B 0,C 180,E1 -696.589,E2 -696.589} C_VEL
LIN {X 0,Y 601.43,Z 304.573,A -85,B 0,C 180,E1 -699.478,E2 -699.478} C_VEL
LIN {X 0,Y 601.394,Z 304.57,A -85,B 0,C 180,E1 -702.311,E2 -702.311} C_VEL
LIN {X 0,Y 601.403,Z 304.573,A -85,B 0,C 180,E1 -704.408,E2 -704.408} C_VEL
LIN {X 0,Y 601.361,Z 304.574,A -85,B 0,C 180,E1 -707.17,E2 -707.17} C_VEL
LIN {X 0,Y 601.433,Z 304.571,A -85,B 0,C 180,E1 -709.905,E2 -709.905} C_VEL
LIN {X 0,Y 601.435,Z 304.565,A -85,B 0,C 180,E1 -712.615,E2 -712.615} C_VEL
LIN {X 0,Y 601.409,Z 304.57,A -85,B 0,C 180,E1 -715.308,E2 -715.308} C_VEL
LIN {X 0,Y 601.434,Z 304.567,A -85,B 0,C 180,E1 -717.991,E2 -717.991} C_VEL
LIN {X 0,Y 601.411,Z 304.568,A -85,B 0,C 180,E1 -720.67,E2 -720.67} C_VEL
LIN {X 0,Y 601.422,Z 304.572,A -85,B 0,C 180,E1 -723.35,E2 -723.35} C_VEL
LIN {X 0,Y 601.44,Z 304.564,A -85,B 0,C 180,E1 -726.037,E2 -726.037} C_VEL
LIN {X 0,Y 601.436,Z 304.57,A -85,B 0,C 180,E1 -728.738,E2 -728.738} C_VEL
LIN {X 0,Y 601.405,Z 304.569,A -85,B 0,C 180,E1 -731.459,E2 -731.459} C_VEL
LIN {X 0,Y 601.397,Z 304.571,A -85,B 0,C 180,E1 -734.206,E2 -734.206} C_VEL
LIN {X 0,Y 601.405,Z 304.573,A -85,B 0,C 180,E1 -736.987,E2 -736.987} C_VEL
LIN {X 0,Y 601.404,Z 304.568,A -85,B 0,C 180,E1 -739.81,E2 -739.81} C_VEL
LIN {X 0,Y 601.41,Z 304.571,A -85,B 0,C 180,E1 -742.606,E2 -742.606} C_VEL
LIN {X 0,Y 601.391,Z 304.57,A -85,B 0,C 180,E1 -744.879,E2 -744.879} C_VEL
LIN {X 0,Y 601.397,Z 304.576,A -85,B 0,C 180,E1 -747.36,E2 -747.36} C_VEL
LIN {X 0,Y 601.394,Z 304.57,A -85,B 0,C 180,E1 -750.166,E2 -750.166} C_VEL
LIN {X 0,Y 601.42,Z 304.572,A -85,B 0,C 180,E1 -752.716,E2 -752.716} C_VEL
LIN {X 0,Y 601.394,Z 304.57,A -85,B 0,C 180,E1 -755.113,E2 -755.113} C_VEL
LIN {X 0,Y 601.433,Z 304.568,A -85,B 0,C 180,E1 -757.419,E2 -757.419} C_VEL
LIN {X 0,Y 601.375,Z 304.573,A -85,B 0,C 180,E1 -759.998,E2 -759.998} C_VEL
LIN {X 0,Y 601.379,Z 304.576,A -85,B 0,C 180,E1 -762.673,E2 -762.673} C_VEL
LIN {X 0,Y 601.396,Z 304.569,A -85,B 0,C 180,E1 -765.48,E2 -765.48} C_VEL
LIN {X 0,Y 601.424,Z 304.568,A -85,B 0,C 180,E1 -768.407,E2 -768.407} C_VEL
LIN {X 0,Y 601.41,Z 304.569,A -85,B 0,C 180,E1 -770.874,E2 -770.874} C_VEL
LIN {X 0,Y 601.398,Z 304.575,A -85,B 0,C 180,E1 -773.417,E2 -773.417} C_VEL
LIN {X 0,Y 601.427,Z 304.725,A -85,B 0,C 180,E1 -774.335,E2 -774.335} C_VEL
LIN {X 0,Y 601.518,Z 311.17,A -85,B 0,C 180,E1 -776.693,E2 -776.693} C_VEL
LIN {X 0,Y 601.445,Z 318.961,A -85,B 0,C 180,E1 -779.449,E2 -779.449} C_VEL
LIN {X 0,Y 601.447,Z 326.753,A -85,B 0,C 180,E1 -782.134,E2 -782.134} C_VEL
LIN {X 0,Y 601.414,Z 335.657,A -85,B 0,C 180,E1 -785.122,E2 -785.122} C_VEL
LIN {X 0,Y 601.418,Z 342.572,A -85,B 0,C 180,E1 -787.395,E2 -787.395} C_VEL
LIN {X 0,Y 601.409,Z 351.239,A -85,B 0,C 180,E1 -790.191,E2 -790.191} C_VEL
LIN {X 0,Y 601.375,Z 360.144,A -85,B 0,C 180,E1 -793.013,E2 -793.013} C_VEL
LIN {X 0,Y 601.355,Z 369.048,A -85,B 0,C 180,E1 -795.793,E2 -795.793} C_VEL
LIN {X 0,Y 601.372,Z 376.491,A -85,B 0,C 180,E1 -798.092,E2 -798.092} C_VEL
LIN {X 0,Y 601.607,Z 383.509,A -85,B 0,C 180,E1 -798.225,E2 -798.225} C_VEL
LIN {X 0,Y 601.556,Z 395.877,A -85,B 0,C 180,E1 -798.544,E2 -798.544} C_VEL
LIN {X 0,Y 601.494,Z 408.836,A -85,B 0,C 180,E1 -799.027,E2 -799.027} C_VEL
LIN {X 0,Y 601.453,Z 421.326,A -85,B 0,C 180,E1 -799.65,E2 -799.65} C_VEL
LIN {X 0,Y 601.467,Z 431.929,A -85,B 0,C 180,E1 -800.33,E2 -800.33} C_VEL
LIN {X 0,Y 601.435,Z 441.597,A -85,B 0,C 180,E1 -801.093,E2 -801.093} C_VEL
LIN {X 0,Y 601.407,Z 450.412,A -85,B 0,C 180,E1 -801.939,E2 -801.939} C_VEL
LIN {X 0,Y 601.388,Z 457.689,A -85,B 0,C 180,E1 -802.783,E2 -802.783} C_VEL
LIN {X 0,Y 601.375,Z 464.773,A -85,B 0,C 180,E1 -803.782,E2 -803.782} C_VEL
LIN {X 0,Y 601.373,Z 469.679,A -85,B 0,C 180,E1 -804.635,E2 -804.635} C_VEL
LIN {X 0,Y 601.354,Z 474.37,A -85,B 0,C 180,E1 -805.643,E2 -805.643} C_VEL
LIN {X 0,Y 601.344,Z 477.955,A -85,B 0,C 180,E1 -806.65,E2 -806.65} C_VEL
LIN {X 0,Y 601.325,Z 479.808,A -85,B 0,C 180,E1 -807.32,E2 -807.32} C_VEL
LIN {X 0,Y 601.343,Z 481.201,A -85,B 0,C 180,E1 -807.99,E2 -807.99} C_VEL
LIN {X 0,Y 601.339,Z 482.783,A -85,B 0,C 180,E1 -809.33,E2 -809.33} C_VEL
LIN {X 0,Y 601.335,Z 483,A -85,B 0,C 180,E1 -810,E2 -810} C_VEL
LIN {X 0,Y 601.347,Z 482.184,A -85,B 0,C 180,E1 -811.339,E2 -811.339} C_VEL
LIN {X 0,Y 601.343,Z 481.202,A -85,B 0,C 180,E1 -812.009,E2 -812.009} C_VEL
LIN {X 0,Y 601.325,Z 479.81,A -85,B 0,C 180,E1 -812.679,E2 -812.679} C_VEL
LIN {X 0,Y 601.368,Z 476.897,A -85,B 0,C 180,E1 -813.685,E2 -813.685} C_VEL
LIN {X 0,Y 601.336,Z 472.952,A -85,B 0,C 180,E1 -814.692,E2 -814.692} C_VEL
LIN {X 0,Y 601.373,Z 466.879,A -85,B 0,C 180,E1 -815.869,E2 -815.869} C_VEL
LIN {X 0,Y 601.381,Z 460.238,A -85,B 0,C 180,E1 -816.879,E2 -816.879} C_VEL
LIN {X 0,Y 601.4,Z 451.993,A -85,B 0,C 180,E1 -817.892,E2 -817.892} C_VEL
LIN {X 0,Y 601.436,Z 443.542,A -85,B 0,C 180,E1 -818.737,E2 -818.737} C_VEL
LIN {X 0,Y 601.449,Z 433.098,A -85,B 0,C 180,E1 -819.585,E2 -819.585} C_VEL
LIN {X 0,Y 601.478,Z 422.764,A -85,B 0,C 180,E1 -820.264,E2 -820.264} C_VEL
LIN {X 0,Y 601.482,Z 411.238,A -85,B 0,C 180,E1 -820.868,E2 -820.868} C_VEL
LIN {X 0,Y 601.526,Z 398.35,A -85,B 0,C 180,E1 -821.375,E2 -821.375} C_VEL
LIN {X 0,Y 601.611,Z 385.461,A -85,B 0,C 180,E1 -821.732,E2 -821.732} C_VEL
LIN {X 0,Y 601.503,Z 377.652,A -85,B 0,C 180,E1 -821.884,E2 -821.884} C_VEL
LIN {X 0,Y 601.344,Z 376.424,A -85,B 0,C 180,E1 -821.929,E2 -821.929} C_VEL
LIN {X 0,Y 601.348,Z 367.937,A -85,B 0,C 180,E1 -824.552,E2 -824.552} C_VEL
LIN {X 0,Y 601.396,Z 359.033,A -85,B 0,C 180,E1 -827.337,E2 -827.337} C_VEL
LIN {X 0,Y 601.393,Z 350.128,A -85,B 0,C 180,E1 -830.165,E2 -830.165} C_VEL
LIN {X 0,Y 601.413,Z 342.337,A -85,B 0,C 180,E1 -832.682,E2 -832.682} C_VEL
LIN {X 0,Y 601.407,Z 334.546,A -85,B 0,C 180,E1 -835.247,E2 -835.247} C_VEL
LIN {X 0,Y 601.446,Z 326.755,A -85,B 0,C 180,E1 -837.865,E2 -837.865} C_VEL
LIN {X 0,Y 601.445,Z 318.963,A -85,B 0,C 180,E1 -840.55,E2 -840.55} C_VEL
LIN {X 0,Y 601.517,Z 311.172,A -85,B 0,C 180,E1 -843.307,E2 -843.307} C_VEL
LIN {X 0,Y 601.399,Z 304.574,A -85,B 0,C 180,E1 -845.731,E2 -845.731} C_VEL
LIN {X 0,Y 601.422,Z 304.573,A -85,B 0,C 180,E1 -848.469,E2 -848.469} C_VEL
LIN {X 0,Y 601.416,Z 304.568,A -85,B 0,C 180,E1 -850.873,E2 -850.873} C_VEL
LIN {X 0,Y 601.444,Z 304.569,A -85,B 0,C 180,E1 -853.583,E2 -853.583} C_VEL
LIN {X 0,Y 601.421,Z 304.566,A -85,B 0,C 180,E1 -856.427,E2 -856.427} C_VEL
LIN {X 0,Y 601.396,Z 304.57,A -85,B 0,C 180,E1 -859.427,E2 -859.427} C_VEL
LIN {X 0,Y 601.402,Z 304.569,A -85,B 0,C 180,E1 -861.73,E2 -861.73} C_VEL
LIN {X 0,Y 601.401,Z 304.573,A -85,B 0,C 180,E1 -864.246,E2 -864.246} C_VEL
LIN {X 0,Y 601.424,Z 304.566,A -85,B 0,C 180,E1 -866.686,E2 -866.686} C_VEL
LIN {X 0,Y 601.415,Z 304.574,A -85,B 0,C 180,E1 -869.058,E2 -869.058} C_VEL
LIN {X 0,Y 601.392,Z 304.571,A -85,B 0,C 180,E1 -871.371,E2 -871.371} C_VEL
LIN {X 0,Y 601.407,Z 304.573,A -85,B 0,C 180,E1 -874.131,E2 -874.131} C_VEL
LIN {X 0,Y 601.416,Z 304.568,A -85,B 0,C 180,E1 -876.589,E2 -876.589} C_VEL
LIN {X 0,Y 601.428,Z 304.573,A -85,B 0,C 180,E1 -879.478,E2 -879.478} C_VEL
LIN {X 0,Y 601.392,Z 304.571,A -85,B 0,C 180,E1 -882.311,E2 -882.311} C_VEL
LIN {X 0,Y 601.399,Z 304.574,A -85,B 0,C 180,E1 -884.408,E2 -884.408} C_VEL
LIN {X 0,Y 601.381,Z 304.571,A -85,B 0,C 180,E1 -887.171,E2 -887.171} C_VEL
LIN {X 0,Y 601.433,Z 304.57,A -85,B 0,C 180,E1 -889.905,E2 -889.905} C_VEL
LIN {X 0,Y 601.445,Z 304.564,A -85,B 0,C 180,E1 -892.615,E2 -892.615} C_VEL
LIN {X 0,Y 601.407,Z 304.57,A -85,B 0,C 180,E1 -895.308,E2 -895.308} C_VEL
LIN {X 0,Y 601.434,Z 304.568,A -85,B 0,C 180,E1 -897.991,E2 -897.991} C_VEL
LIN {X 0,Y 601.408,Z 304.568,A -85,B 0,C 180,E1 -900.67,E2 -900.67} C_VEL
LIN {X 0,Y 601.422,Z 304.573,A -85,B 0,C 180,E1 -903.35,E2 -903.35} C_VEL
LIN {X 0,Y 601.44,Z 304.564,A -85,B 0,C 180,E1 -906.037,E2 -906.037} C_VEL
LIN {X 0,Y 601.432,Z 304.57,A -85,B 0,C 180,E1 -908.738,E2 -908.738} C_VEL
LIN {X 0,Y 601.402,Z 304.57,A -85,B 0,C 180,E1 -911.459,E2 -911.459} C_VEL
LIN {X 0,Y 601.388,Z 304.573,A -85,B 0,C 180,E1 -912.382,E2 -912.382} C_VEL
LIN {X 0,Y 600.705,Z 304.656,A -85,B 0,C 180,E1 -912.941,E2 -912.941} C_VEL
LIN {X 0,Y 597.844,Z 305.017,A -85,B 0,C 180,E1 -913.849,E2 -913.849} C_VEL
LIN {X 0,Y 595.439,Z 305.316,A -85,B 0,C 180,E1 -914.579,E2 -914.579} C_VEL
LIN {X 0,Y 594.412,Z 305.443,A -85,B 0,C 180,E1 -915.143,E2 -915.143} C_VEL
LIN {X 0,Y 594.331,Z 305.451,A -85,B 0,C 180,E1 -915.334,E2 -915.334} C_VEL
LIN {X 0,Y 594.37,Z 305.444,A -85,B 0,C 180,E1 -917.905,E2 -917.905} C_VEL
LIN {X 0,Y 594.377,Z 305.447,A -85,B 0,C 180,E1 -920.919,E2 -920.919} C_VEL
LIN {X 0,Y 594.386,Z 305.446,A -85,B 0,C 180,E1 -923.704,E2 -923.704} C_VEL
LIN {X 0,Y 594.356,Z 305.45,A -85,B 0,C 180,E1 -926.02,E2 -926.02} C_VEL
LIN {X 0,Y 594.315,Z 305.451,A -85,B 0,C 180,E1 -928.23,E2 -928.23} C_VEL
LIN {X 0,Y 594.366,Z 305.448,A -85,B 0,C 180,E1 -930.561,E2 -930.561} C_VEL
LIN {X 0,Y 594.372,Z 305.447,A -85,B 0,C 180,E1 -932.951,E2 -932.951} C_VEL
LIN {X 0,Y 594.375,Z 305.445,A -85,B 0,C 180,E1 -935.407,E2 -935.407} C_VEL
LIN {X 0,Y 594.373,Z 305.449,A -85,B 0,C 180,E1 -937.942,E2 -937.942} C_VEL
LIN {X 0,Y 594.363,Z 305.449,A -85,B 0,C 180,E1 -940.822,E2 -940.822} C_VEL
LIN {X 0,Y 594.345,Z 305.448,A -85,B 0,C 180,E1 -943.839,E2 -943.839} C_VEL
LIN {X 0,Y 594.362,Z 305.447,A -85,B 0,C 180,E1 -946.702,E2 -946.702} C_VEL
LIN {X 0,Y 594.369,Z 305.449,A -85,B 0,C 180,E1 -949.434,E2 -949.434} C_VEL
LIN {X 0,Y 594.383,Z 305.443,A -85,B 0,C 180,E1 -952.393,E2 -952.393} C_VEL
LIN {X 0,Y 594.295,Z 305.471,A -85,B 0,C 180,E1 -954.685,E2 -954.685} C_VEL
LIN {X 0,Y 594.372,Z 309.504,A -85,B 0,C 180,E1 -957.09,E2 -957.09} C_VEL
LIN {X 0,Y 594.327,Z 313.924,A -85,B 0,C 180,E1 -959.682,E2 -959.682} C_VEL
LIN {X 0,Y 594.331,Z 318.902,A -85,B 0,C 180,E1 -962.538,E2 -962.538} C_VEL
LIN {X 0,Y 594.294,Z 323.04,A -85,B 0,C 180,E1 -964.804,E2 -964.804} C_VEL
LIN {X 0,Y 594.273,Z 328.569,A -85,B 0,C 180,E1 -967.764,E2 -967.764} C_VEL
LIN {X 0,Y 594.242,Z 332.716,A -85,B 0,C 180,E1 -969.942,E2 -969.942} C_VEL
LIN {X 0,Y 594.241,Z 336.863,A -85,B 0,C 180,E1 -972.092,E2 -972.092} C_VEL
LIN {X 0,Y 594.255,Z 342.393,A -85,B 0,C 180,E1 -974.92,E2 -974.92} C_VEL
LIN {X 0,Y 594.274,Z 348.441,A -85,B 0,C 180,E1 -977.97,E2 -977.97} C_VEL
LIN {X 0,Y 594.291,Z 348.884,A -85,B 0,C 180,E1 -978.035,E2 -978.035} C_VEL
LIN {X 0,Y 594.647,Z 354.47,A -85,B 0,C 180,E1 -978.15,E2 -978.15} C_VEL
LIN {X 0,Y 594.566,Z 367.158,A -85,B 0,C 180,E1 -978.495,E2 -978.495} C_VEL
LIN {X 0,Y 594.501,Z 379.759,A -85,B 0,C 180,E1 -978.982,E2 -978.982} C_VEL
LIN {X 0,Y 594.467,Z 390.534,A -85,B 0,C 180,E1 -979.528,E2 -979.528} C_VEL
LIN {X 0,Y 594.449,Z 401.323,A -85,B 0,C 180,E1 -980.216,E2 -980.216} C_VEL
LIN {X 0,Y 594.404,Z 411.096,A -85,B 0,C 180,E1 -980.987,E2 -980.987} C_VEL
LIN {X 0,Y 594.366,Z 419.99,A -85,B 0,C 180,E1 -981.843,E2 -981.843} C_VEL
LIN {X 0,Y 594.345,Z 428.675,A -85,B 0,C 180,E1 -982.868,E2 -982.868} C_VEL
LIN {X 0,Y 594.29,Z 435.602,A -85,B 0,C 180,E1 -983.891,E2 -983.891} C_VEL
LIN {X 0,Y 594.253,Z 441.153,A -85,B 0,C 180,E1 -984.912,E2 -984.912} C_VEL
LIN {X 0,Y 594.263,Z 445.515,A -85,B 0,C 180,E1 -985.931,E2 -985.931} C_VEL
LIN {X 0,Y 594.267,Z 447.818,A -85,B 0,C 180,E1 -986.61,E2 -986.61} C_VEL
LIN {X 0,Y 594.225,Z 449.695,A -85,B 0,C 180,E1 -987.289,E2 -987.289} C_VEL
LIN {X 0,Y 594.242,Z 451.128,A -85,B 0,C 180,E1 -987.967,E2 -987.967} C_VEL
LIN {X 0,Y 594.24,Z 452.753,A -85,B 0,C 180,E1 -989.323,E2 -989.323} C_VEL
LIN {X 0,Y 594.236,Z 452.996,A -85,B 0,C 180,E1 -990,E2 -990} C_VEL
LIN {X 0,Y 594.239,Z 452.815,A -85,B 0,C 180,E1 -990.678,E2 -990.678} C_VEL
LIN {X 0,Y 594.242,Z 451.274,A -85,B 0,C 180,E1 -992.034,E2 -992.034} C_VEL
LIN {X 0,Y 594.226,Z 449.914,A -85,B 0,C 180,E1 -992.712,E2 -992.712} C_VEL
LIN {X 0,Y 594.289,Z 447.037,A -85,B 0,C 180,E1 -993.73,E2 -993.73} C_VEL
LIN {X 0,Y 594.242,Z 443.137,A -85,B 0,C 180,E1 -994.749,E2 -994.749} C_VEL
LIN {X 0,Y 594.3,Z 438.106,A -85,B 0,C 180,E1 -995.769,E2 -995.769} C_VEL
LIN {X 0,Y 594.316,Z 431.786,A -85,B 0,C 180,E1 -996.791,E2 -996.791} C_VEL
LIN {X 0,Y 594.346,Z 423.868,A -85,B 0,C 180,E1 -997.816,E2 -997.816} C_VEL
LIN {X 0,Y 594.381,Z 414.022,A -85,B 0,C 180,E1 -998.842,E2 -998.842} C_VEL
LIN {X 0,Y 594.431,Z 403.701,A -85,B 0,C 180,E1 -999.699,E2 -999.699} C_VEL
LIN {X 0,Y 594.464,Z 392.077,A -85,B 0,C 180,E1 -1000.473,E2 -1000.473} C_VEL
LIN {X 0,Y 594.504,Z 380.934,A -85,B 0,C 180,E1 -1001.057,E2 -1001.057} C_VEL
LIN {X 0,Y 594.585,Z 368.551,A -85,B 0,C 180,E1 -1001.548,E2 -1001.548} C_VEL
LIN {X 0,Y 594.666,Z 355.51,A -85,B 0,C 180,E1 -1001.915,E2 -1001.915} C_VEL
LIN {X 0,Y 594.484,Z 350.174,A -85,B 0,C 180,E1 -1002.027,E2 -1002.027} C_VEL
LIN {X 0,Y 594.247,Z 348.533,A -85,B 0,C 180,E1 -1002.075,E2 -1002.075} C_VEL
LIN {X 0,Y 594.253,Z 342.569,A -85,B 0,C 180,E1 -1005.081,E2 -1005.081} C_VEL
LIN {X 0,Y 594.231,Z 337.037,A -85,B 0,C 180,E1 -1007.909,E2 -1007.909} C_VEL
LIN {X 0,Y 594.298,Z 331.504,A -85,B 0,C 180,E1 -1010.779,E2 -1010.779} C_VEL
LIN {X 0,Y 594.28,Z 325.972,A -85,B 0,C 180,E1 -1013.709,E2 -1013.709} C_VEL
LIN {X 0,Y 594.298,Z 321.717,A -85,B 0,C 180,E1 -1016.005,E2 -1016.005} C_VEL
LIN {X 0,Y 594.302,Z 317.691,A -85,B 0,C 180,E1 -1018.231,E2 -1018.231} C_VEL
LIN {X 0,Y 594.301,Z 313.64,A -85,B 0,C 180,E1 -1020.564,E2 -1020.564} C_VEL
LIN {X 0,Y 594.372,Z 309.589,A -85,B 0,C 180,E1 -1022.95,E2 -1022.95} C_VEL
LIN {X 0,Y 594.296,Z 305.459,A -85,B 0,C 180,E1 -1025.412,E2 -1025.412} C_VEL
LIN {X 0,Y 594.372,Z 305.445,A -85,B 0,C 180,E1 -1027.941,E2 -1027.941} C_VEL
LIN {X 0,Y 594.377,Z 305.446,A -85,B 0,C 180,E1 -1030.822,E2 -1030.822} C_VEL
LIN {X 0,Y 594.367,Z 305.446,A -85,B 0,C 180,E1 -1033.299,E2 -1033.299} C_VEL
LIN {X 0,Y 594.349,Z 305.447,A -85,B 0,C 180,E1 -1036.162,E2 -1036.162} C_VEL
LIN {X 0,Y 594.366,Z 305.45,A -85,B 0,C 180,E1 -1039.179,E2 -1039.179} C_VEL
LIN {X 0,Y 594.372,Z 305.448,A -85,B 0,C 180,E1 -1042.058,E2 -1042.058} C_VEL
LIN {X 0,Y 594.353,Z 305.448,A -85,B 0,C 180,E1 -1044.675,E2 -1044.675} C_VEL
LIN {X 0,Y 594.378,Z 305.446,A -85,B 0,C 180,E1 -1047.088,E2 -1047.088} C_VEL
LIN {X 0,Y 594.364,Z 305.447,A -85,B 0,C 180,E1 -1049.674,E2 -1049.674} C_VEL
LIN {X 0,Y 594.352,Z 305.453,A -85,B 0,C 180,E1 -1052.538,E2 -1052.538} C_VEL
LIN {X 0,Y 594.368,Z 305.447,A -85,B 0,C 180,E1 -1054.806,E2 -1054.806} C_VEL
LIN {X 0,Y 594.359,Z 305.447,A -85,B 0,C 180,E1 -1057.264,E2 -1057.264} C_VEL
LIN {X 0,Y 594.374,Z 305.446,A -85,B 0,C 180,E1 -1059.946,E2 -1059.946} C_VEL
LIN {X 0,Y 594.374,Z 305.45,A -85,B 0,C 180,E1 -1062.806,E2 -1062.806} C_VEL
LIN {X 0,Y 594.367,Z 305.446,A -85,B 0,C 180,E1 -1065.832,E2 -1065.832} C_VEL
LIN {X 0,Y 594.37,Z 305.448,A -85,B 0,C 180,E1 -1068.404,E2 -1068.404} C_VEL
LIN {X 0,Y 594.392,Z 305.445,A -85,B 0,C 180,E1 -1071.158,E2 -1071.158} C_VEL
LIN {X 0,Y 594.391,Z 305.442,A -85,B 0,C 180,E1 -1073.891,E2 -1073.891} C_VEL
LIN {X 0,Y 594.378,Z 305.451,A -85,B 0,C 180,E1 -1076.611,E2 -1076.611} C_VEL
LIN {X 0,Y 594.386,Z 305.443,A -85,B 0,C 180,E1 -1079.322,E2 -1079.322} C_VEL
LIN {X 0,Y 594.401,Z 305.445,A -85,B 0,C 180,E1 -1082.033,E2 -1082.033} C_VEL
LIN {X 0,Y 594.377,Z 305.446,A -85,B 0,C 180,E1 -1084.748,E2 -1084.748} C_VEL
LIN {X 0,Y 594.39,Z 305.443,A -85,B 0,C 180,E1 -1087.473,E2 -1087.473} C_VEL
LIN {X 0,Y 594.391,Z 305.448,A -85,B 0,C 180,E1 -1090.216,E2 -1090.216} C_VEL
LIN {X 0,Y 594.319,Z 305.451,A -85,B 0,C 180,E1 -1092.984,E2 -1092.984} C_VEL
LIN {X 0,Y 594.348,Z 305.451,A -85,B 0,C 180,E1 -1095.781,E2 -1095.781} C_VEL
LIN {X 0,Y 594.377,Z 305.448,A -85,B 0,C 180,E1 -1098.618,E2 -1098.618} C_VEL
LIN {X 0,Y 594.367,Z 305.445,A -85,B 0,C 180,E1 -1101.503,E2 -1101.503} C_VEL
LIN {X 0,Y 594.384,Z 305.445,A -85,B 0,C 180,E1 -1104.446,E2 -1104.446} C_VEL
LIN {X 0,Y 594.356,Z 305.446,A -85,B 0,C 180,E1 -1106.701,E2 -1106.701} C_VEL
LIN {X 0,Y 594.347,Z 305.448,A -85,B 0,C 180,E1 -1109.778,E2 -1109.778} C_VEL
LIN {X 0,Y 594.366,Z 305.447,A -85,B 0,C 180,E1 -1112.147,E2 -1112.147} C_VEL
LIN {X 0,Y 594.377,Z 305.447,A -85,B 0,C 180,E1 -1114.58,E2 -1114.58} C_VEL
LIN {X 0,Y 594.383,Z 305.443,A -85,B 0,C 180,E1 -1117.087,E2 -1117.087} C_VEL
LIN {X 0,Y 594.34,Z 305.451,A -85,B 0,C 180,E1 -1119.771,E2 -1119.771} C_VEL
LIN {X 0,Y 594.337,Z 305.45,A -85,B 0,C 180,E1 -1122.378,E2 -1122.378} C_VEL
LIN {X 0,Y 594.354,Z 305.447,A -85,B 0,C 180,E1 -1125.193,E2 -1125.193} C_VEL
LIN {X 0,Y 594.384,Z 305.449,A -85,B 0,C 180,E1 -1128.152,E2 -1128.152} C_VEL
LIN {X 0,Y 594.371,Z 305.449,A -85,B 0,C 180,E1 -1131.194,E2 -1131.194} C_VEL
LIN {X 0,Y 594.346,Z 305.451,A -85,B 0,C 180,E1 -1133.965,E2 -1133.965} C_VEL
LIN {X 0,Y 594.366,Z 305.605,A -85,B 0,C 180,E1 -1134.176,E2 -1134.176} C_VEL
LIN {X 0,Y 594.472,Z 308.944,A -85,B 0,C 180,E1 -1135.427,E2 -1135.427} C_VEL
LIN {X 0,Y 594.451,Z 314.533,A -85,B 0,C 180,E1 -1137.466,E2 -1137.466} C_VEL
LIN {X 0,Y 594.454,Z 322.3,A -85,B 0,C 180,E1 -1140.228,E2 -1140.228} C_VEL
LIN {X 0,Y 594.402,Z 330.092,A -85,B 0,C 180,E1 -1142.922,E2 -1142.922} C_VEL
LIN {X 0,Y 594.401,Z 337.912,A -85,B 0,C 180,E1 -1145.564,E2 -1145.564} C_VEL
LIN {X 0,Y 594.386,Z 346.787,A -85,B 0,C 180,E1 -1148.498,E2 -1148.498} C_VEL
LIN {X 0,Y 594.325,Z 355.692,A -85,B 0,C 180,E1 -1151.381,E2 -1151.381} C_VEL
LIN {X 0,Y 594.303,Z 364.596,A -85,B 0,C 180,E1 -1154.217,E2 -1154.217} C_VEL
LIN {X 0,Y 594.273,Z 373.5,A -85,B 0,C 180,E1 -1157.015,E2 -1157.015} C_VEL
LIN {X 0,Y 594.28,Z 376.491,A -85,B 0,C 180,E1 -1157.948,E2 -1157.948} C_VEL
LIN {X 0,Y 594.669,Z 381.226,A -85,B 0,C 180,E1 -1158.042,E2 -1158.042} C_VEL
LIN {X 0,Y 594.612,Z 394.493,A -85,B 0,C 180,E1 -1158.365,E2 -1158.365} C_VEL
LIN {X 0,Y 594.531,Z 406.66,A -85,B 0,C 180,E1 -1158.802,E2 -1158.802} C_VEL
LIN {X 0,Y 594.476,Z 418.206,A -85,B 0,C 180,E1 -1159.355,E2 -1159.355} C_VEL
LIN {X 0,Y 594.465,Z 429.474,A -85,B 0,C 180,E1 -1160.043,E2 -1160.043} C_VEL
LIN {X 0,Y 594.406,Z 439.645,A -85,B 0,C 180,E1 -1160.815,E2 -1160.815} C_VEL
LIN {X 0,Y 594.372,Z 448.786,A -85,B 0,C 180,E1 -1161.671,E2 -1161.671} C_VEL
LIN {X 0,Y 594.317,Z 457.689,A -85,B 0,C 180,E1 -1162.697,E2 -1162.697} C_VEL
LIN {X 0,Y 594.281,Z 464.168,A -85,B 0,C 180,E1 -1163.615,E2 -1163.615} C_VEL
LIN {X 0,Y 594.289,Z 469.679,A -85,B 0,C 180,E1 -1164.571,E2 -1164.571} C_VEL
LIN {X 0,Y 594.27,Z 474.37,A -85,B 0,C 180,E1 -1165.591,E2 -1165.591} C_VEL
LIN {X 0,Y 594.267,Z 477.955,A -85,B 0,C 180,E1 -1166.61,E2 -1166.61} C_VEL
LIN {X 0,Y 594.226,Z 479.808,A -85,B 0,C 180,E1 -1167.288,E2 -1167.288} C_VEL
LIN {X 0,Y 594.242,Z 481.201,A -85,B 0,C 180,E1 -1167.966,E2 -1167.966} C_VEL
LIN {X 0,Y 594.239,Z 482.784,A -85,B 0,C 180,E1 -1169.322,E2 -1169.322} C_VEL
LIN {X 0,Y 594.236,Z 483,A -85,B 0,C 180,E1 -1170,E2 -1170} C_VEL
LIN {X 0,Y 594.247,Z 482.185,A -85,B 0,C 180,E1 -1171.355,E2 -1171.355} C_VEL
LIN {X 0,Y 594.242,Z 481.202,A -85,B 0,C 180,E1 -1172.033,E2 -1172.033} C_VEL
LIN {X 0,Y 594.226,Z 479.81,A -85,B 0,C 180,E1 -1172.711,E2 -1172.711} C_VEL
LIN {X 0,Y 594.289,Z 476.897,A -85,B 0,C 180,E1 -1173.729,E2 -1173.729} C_VEL
LIN {X 0,Y 594.241,Z 472.951,A -85,B 0,C 180,E1 -1174.748,E2 -1174.748} C_VEL
LIN {X 0,Y 594.305,Z 466.879,A -85,B 0,C 180,E1 -1175.939,E2 -1175.939} C_VEL
LIN {X 0,Y 594.307,Z 460.239,A -85,B 0,C 180,E1 -1176.962,E2 -1176.962} C_VEL
LIN {X 0,Y 594.359,Z 451.993,A -85,B 0,C 180,E1 -1177.986,E2 -1177.986} C_VEL
LIN {X 0,Y 594.382,Z 443.542,A -85,B 0,C 180,E1 -1178.842,E2 -1178.842} C_VEL
LIN {X 0,Y 594.431,Z 433.098,A -85,B 0,C 180,E1 -1179.699,E2 -1179.699} C_VEL
LIN {X 0,Y 594.454,Z 422.765,A -85,B 0,C 180,E1 -1180.386,E2 -1180.386} C_VEL
LIN {X 0,Y 594.5,Z 410.782,A -85,B 0,C 180,E1 -1181.018,E2 -1181.018} C_VEL
LIN {X 0,Y 594.559,Z 398.506,A -85,B 0,C 180,E1 -1181.505,E2 -1181.505} C_VEL
LIN {X 0,Y 594.681,Z 385.461,A -85,B 0,C 180,E1 -1181.87,E2 -1181.87} C_VEL
LIN {X 0,Y 594.42,Z 377.651,A -85,B 0,C 180,E1 -1182.027,E2 -1182.027} C_VEL
LIN {X 0,Y 594.286,Z 376.424,A -85,B 0,C 180,E1 -1182.073,E2 -1182.073} C_VEL
LIN {X 0,Y 594.295,Z 367.937,A -85,B 0,C 180,E1 -1184.729,E2 -1184.729} C_VEL
LIN {X 0,Y 594.328,Z 359.033,A -85,B 0,C 180,E1 -1187.549,E2 -1187.549} C_VEL
LIN {X 0,Y 594.361,Z 350.128,A -85,B 0,C 180,E1 -1190.415,E2 -1190.415} C_VEL
LIN {X 0,Y 594.375,Z 342.337,A -85,B 0,C 180,E1 -1192.966,E2 -1192.966} C_VEL
LIN {X 0,Y 594.403,Z 334.546,A -85,B 0,C 180,E1 -1195.566,E2 -1195.566} C_VEL
LIN {X 0,Y 594.421,Z 326.755,A -85,B 0,C 180,E1 -1198.224,E2 -1198.224} C_VEL
LIN {X 0,Y 594.446,Z 320.076,A -85,B 0,C 180,E1 -1200.555,E2 -1200.555} C_VEL
LIN {X 0,Y 594.533,Z 312.285,A -85,B 0,C 180,E1 -1203.344,E2 -1203.344} C_VEL
LIN {X 0,Y 594.545,Z 306.72,A -85,B 0,C 180,E1 -1205.394,E2 -1205.394} C_VEL
LIN {X 0,Y 594.353,Z 305.452,A -85,B 0,C 180,E1 -1205.929,E2 -1205.929} C_VEL
LIN {X 0,Y 594.382,Z 305.448,A -85,B 0,C 180,E1 -1208.804,E2 -1208.804} C_VEL
LIN {X 0,Y 594.382,Z 305.449,A -85,B 0,C 180,E1 -1211.848,E2 -1211.848} C_VEL
LIN {X 0,Y 594.376,Z 305.445,A -85,B 0,C 180,E1 -1214.235,E2 -1214.235} C_VEL
LIN {X 0,Y 594.353,Z 305.448,A -85,B 0,C 180,E1 -1216.699,E2 -1216.699} C_VEL
LIN {X 0,Y 594.35,Z 305.448,A -85,B 0,C 180,E1 -1219.431,E2 -1219.431} C_VEL
LIN {X 0,Y 594.382,Z 305.45,A -85,B 0,C 180,E1 -1222.391,E2 -1222.391} C_VEL
LIN {X 0,Y 594.377,Z 305.444,A -85,B 0,C 180,E1 -1224.671,E2 -1224.671} C_VEL
LIN {X 0,Y 594.373,Z 305.447,A -85,B 0,C 180,E1 -1227.087,E2 -1227.087} C_VEL
LIN {X 0,Y 594.359,Z 305.447,A -85,B 0,C 180,E1 -1229.674,E2 -1229.674} C_VEL
LIN {X 0,Y 594.364,Z 305.453,A -85,B 0,C 180,E1 -1232.538,E2 -1232.538} C_VEL
LIN {X 0,Y 594.388,Z 305.444,A -85,B 0,C 180,E1 -1235.563,E2 -1235.563} C_VEL
LIN {X 0,Y 594.365,Z 305.445,A -85,B 0,C 180,E1 -1238.497,E2 -1238.497} C_VEL
LIN {X 0,Y 594.375,Z 305.448,A -85,B 0,C 180,E1 -1241.382,E2 -1241.382} C_VEL
LIN {X 0,Y 594.349,Z 305.45,A -85,B 0,C 180,E1 -1244.219,E2 -1244.219} C_VEL
LIN {X 0,Y 594.356,Z 305.453,A -85,B 0,C 180,E1 -1246.32,E2 -1246.32} C_VEL
LIN {X 0,Y 594.357,Z 305.447,A -85,B 0,C 180,E1 -1249.094,E2 -1249.094} C_VEL
LIN {X 0,Y 594.413,Z 305.441,A -85,B 0,C 180,E1 -1251.843,E2 -1251.843} C_VEL
LIN {X 0,Y 594.4,Z 305.445,A -85,B 0,C 180,E1 -1254.572,E2 -1254.572} C_VEL
LIN {X 0,Y 594.381,Z 305.443,A -85,B 0,C 180,E1 -1257.289,E2 -1257.289} C_VEL
LIN {X 0,Y 594.403,Z 305.448,A -85,B 0,C 180,E1 -1260,E2 -1260} C_VEL
LIN {X 0,Y 594.381,Z 305.443,A -85,B 0,C 180,E1 -1262.711,E2 -1262.711} C_VEL
LIN {X 0,Y 594.4,Z 305.444,A -85,B 0,C 180,E1 -1265.428,E2 -1265.428} C_VEL
LIN {X 0,Y 594.413,Z 305.441,A -85,B 0,C 180,E1 -1268.157,E2 -1268.157} C_VEL
LIN {X 0,Y 594.372,Z 305.444,A -85,B 0,C 180,E1 -1271.072,E2 -1271.072} C_VEL
LIN {X 0,Y 594.357,Z 305.454,A -85,B 0,C 180,E1 -1273.68,E2 -1273.68} C_VEL
LIN {X 0,Y 594.331,Z 305.451,A -85,B 0,C 180,E1 -1275.334,E2 -1275.334} C_VEL
LIN {X 0,Y 593.673,Z 305.534,A -85,B 0,C 180,E1 -1275.9,E2 -1275.9} C_VEL
LIN {X 0,Y 590.827,Z 305.889,A -85,B 0,C 180,E1 -1276.818,E2 -1276.818} C_VEL
LIN {X 0,Y 588.423,Z 306.187,A -85,B 0,C 180,E1 -1277.557,E2 -1277.557} C_VEL
LIN {X 0,Y 587.395,Z 306.314,A -85,B 0,C 180,E1 -1278.127,E2 -1278.127} C_VEL
LIN {X 0,Y 587.314,Z 306.324,A -85,B 0,C 180,E1 -1278.32,E2 -1278.32} C_VEL
LIN {X 0,Y 587.348,Z 306.321,A -85,B 0,C 180,E1 -1281.045,E2 -1281.045} C_VEL
LIN {X 0,Y 587.331,Z 306.329,A -85,B 0,C 180,E1 -1284.007,E2 -1284.007} C_VEL
LIN {X 0,Y 587.318,Z 306.324,A -85,B 0,C 180,E1 -1286.28,E2 -1286.28} C_VEL
LIN {X 0,Y 587.302,Z 306.329,A -85,B 0,C 180,E1 -1289.382,E2 -1289.382} C_VEL
LIN {X 0,Y 587.347,Z 306.319,A -85,B 0,C 180,E1 -1291.838,E2 -1291.838} C_VEL
LIN {X 0,Y 587.348,Z 306.326,A -85,B 0,C 180,E1 -1294.35,E2 -1294.35} C_VEL
LIN {X 0,Y 587.346,Z 306.32,A -85,B 0,C 180,E1 -1296.747,E2 -1296.747} C_VEL
LIN {X 0,Y 587.329,Z 306.329,A -85,B 0,C 180,E1 -1299.361,E2 -1299.361} C_VEL
LIN {X 0,Y 587.295,Z 306.326,A -85,B 0,C 180,E1 -1302.105,E2 -1302.105} C_VEL
LIN {X 0,Y 587.311,Z 306.325,A -85,B 0,C 180,E1 -1305.09,E2 -1305.09} C_VEL
LIN {X 0,Y 587.349,Z 306.326,A -85,B 0,C 180,E1 -1307.929,E2 -1307.929} C_VEL
LIN {X 0,Y 587.329,Z 306.325,A -85,B 0,C 180,E1 -1311.059,E2 -1311.059} C_VEL
LIN {X 0,Y 587.343,Z 306.326,A -85,B 0,C 180,E1 -1313.294,E2 -1313.294} C_VEL
LIN {X 0,Y 587.248,Z 306.335,A -85,B 0,C 180,E1 -1314.47,E2 -1314.47} C_VEL
LIN {X 0,Y 587.284,Z 306.768,A -85,B 0,C 180,E1 -1314.943,E2 -1314.943} C_VEL
LIN {X 0,Y 587.31,Z 310.871,A -85,B 0,C 180,E1 -1317.42,E2 -1317.42} C_VEL
LIN {X 0,Y 587.269,Z 314.945,A -85,B 0,C 180,E1 -1319.827,E2 -1319.827} C_VEL
LIN {X 0,Y 587.222,Z 320.334,A -85,B 0,C 180,E1 -1322.949,E2 -1322.949} C_VEL
LIN {X 0,Y 587.206,Z 324.82,A -85,B 0,C 180,E1 -1325.452,E2 -1325.452} C_VEL
LIN {X 0,Y 587.189,Z 329.953,A -85,B 0,C 180,E1 -1328.221,E2 -1328.221} C_VEL
LIN {X 0,Y 587.208,Z 335.482,A -85,B 0,C 180,E1 -1331.147,E2 -1331.147} C_VEL
LIN {X 0,Y 587.16,Z 341.012,A -85,B 0,C 180,E1 -1334.021,E2 -1334.021} C_VEL
LIN {X 0,Y 587.175,Z 345.159,A -85,B 0,C 180,E1 -1336.15,E2 -1336.15} C_VEL
LIN {X 0,Y 587.151,Z 348.529,A -85,B 0,C 180,E1 -1337.865,E2 -1337.865} C_VEL
LIN {X 0,Y 587.736,Z 353.473,A -85,B 0,C 180,E1 -1337.987,E2 -1337.987} C_VEL
LIN {X 0,Y 587.642,Z 365.965,A -85,B 0,C 180,E1 -1338.317,E2 -1338.317} C_VEL
LIN {X 0,Y 587.559,Z 378.72,A -85,B 0,C 180,E1 -1338.803,E2 -1338.803} C_VEL
LIN {X 0,Y 587.484,Z 390.546,A -85,B 0,C 180,E1 -1339.402,E2 -1339.402} C_VEL
LIN {X 0,Y 587.439,Z 401.329,A -85,B 0,C 180,E1 -1340.098,E2 -1340.098} C_VEL
LIN {X 0,Y 587.357,Z 411.103,A -85,B 0,C 180,E1 -1340.878,E2 -1340.878} C_VEL
LIN {X 0,Y 587.302,Z 419.995,A -85,B 0,C 180,E1 -1341.744,E2 -1341.744} C_VEL
LIN {X 0,Y 587.273,Z 428.679,A -85,B 0,C 180,E1 -1342.782,E2 -1342.782} C_VEL
LIN {X 0,Y 587.214,Z 435.606,A -85,B 0,C 180,E1 -1343.817,E2 -1343.817} C_VEL
LIN {X 0,Y 587.167,Z 441.156,A -85,B 0,C 180,E1 -1344.85,E2 -1344.85} C_VEL
LIN {X 0,Y 587.182,Z 445.517,A -85,B 0,C 180,E1 -1345.882,E2 -1345.882} C_VEL
LIN {X 0,Y 587.193,Z 447.82,A -85,B 0,C 180,E1 -1346.57,E2 -1346.57} C_VEL
LIN {X 0,Y 587.131,Z 449.697,A -85,B 0,C 180,E1 -1347.256,E2 -1347.256} C_VEL
LIN {X 0,Y 587.141,Z 451.128,A -85,B 0,C 180,E1 -1347.942,E2 -1347.942} C_VEL
LIN {X 0,Y 587.14,Z 452.754,A -85,B 0,C 180,E1 -1349.314,E2 -1349.314} C_VEL
LIN {X 0,Y 587.137,Z 452.996,A -85,B 0,C 180,E1 -1350,E2 -1350} C_VEL
LIN {X 0,Y 587.14,Z 452.815,A -85,B 0,C 180,E1 -1350.686,E2 -1350.686} C_VEL
LIN {X 0,Y 587.141,Z 451.273,A -85,B 0,C 180,E1 -1352.058,E2 -1352.058} C_VEL
LIN {X 0,Y 587.133,Z 449.912,A -85,B 0,C 180,E1 -1352.745,E2 -1352.745} C_VEL
LIN {X 0,Y 587.213,Z 447.035,A -85,B 0,C 180,E1 -1353.775,E2 -1353.775} C_VEL
LIN {X 0,Y 587.147,Z 443.135,A -85,B 0,C 180,E1 -1354.807,E2 -1354.807} C_VEL
LIN {X 0,Y 587.23,Z 438.103,A -85,B 0,C 180,E1 -1355.839,E2 -1355.839} C_VEL
LIN {X 0,Y 587.23,Z 431.782,A -85,B 0,C 180,E1 -1356.874,E2 -1356.874} C_VEL
LIN {X 0,Y 587.288,Z 423.864,A -85,B 0,C 180,E1 -1357.91,E2 -1357.91} C_VEL
LIN {X 0,Y 587.343,Z 414.016,A -85,B 0,C 180,E1 -1358.949,E2 -1358.949} C_VEL
LIN {X 0,Y 587.415,Z 403.695,A -85,B 0,C 180,E1 -1359.816,E2 -1359.816} C_VEL
LIN {X 0,Y 587.481,Z 392.066,A -85,B 0,C 180,E1 -1360.599,E2 -1360.599} C_VEL
LIN {X 0,Y 587.515,Z 380.39,A -85,B 0,C 180,E1 -1361.214,E2 -1361.214} C_VEL
LIN {X 0,Y 587.613,Z 368.497,A -85,B 0,C 180,E1 -1361.688,E2 -1361.688} C_VEL
LIN {X 0,Y 587.718,Z 355.486,A -85,B 0,C 180,E1 -1362.058,E2 -1362.058} C_VEL
LIN {X 0,Y 587.519,Z 350.857,A -85,B 0,C 180,E1 -1362.158,E2 -1362.158} C_VEL
LIN {X 0,Y 587.148,Z 348.532,A -85,B 0,C 180,E1 -1362.223,E2 -1362.223} C_VEL
LIN {X 0,Y 587.177,Z 343.951,A -85,B 0,C 180,E1 -1364.558,E2 -1364.558} C_VEL
LIN {X 0,Y 587.141,Z 338.419,A -85,B 0,C 180,E1 -1367.412,E2 -1367.412} C_VEL
LIN {X 0,Y 587.186,Z 334.27,A -85,B 0,C 180,E1 -1369.58,E2 -1369.58} C_VEL
LIN {X 0,Y 587.19,Z 330.12,A -85,B 0,C 180,E1 -1371.779,E2 -1371.779} C_VEL
LIN {X 0,Y 587.205,Z 324.985,A -85,B 0,C 180,E1 -1374.548,E2 -1374.548} C_VEL
LIN {X 0,Y 587.225,Z 320.491,A -85,B 0,C 180,E1 -1377.051,E2 -1377.051} C_VEL
LIN {X 0,Y 587.229,Z 316.44,A -85,B 0,C 180,E1 -1379.386,E2 -1379.386} C_VEL
LIN {X 0,Y 587.314,Z 312.297,A -85,B 0,C 180,E1 -1381.83,E2 -1381.83} C_VEL
LIN {X 0,Y 587.334,Z 308.081,A -85,B 0,C 180,E1 -1384.345,E2 -1384.345} C_VEL
LIN {X 0,Y 587.25,Z 306.335,A -85,B 0,C 180,E1 -1385.531,E2 -1385.531} C_VEL
LIN {X 0,Y 587.329,Z 306.322,A -85,B 0,C 180,E1 -1387.837,E2 -1387.837} C_VEL
LIN {X 0,Y 587.311,Z 306.33,A -85,B 0,C 180,E1 -1390.254,E2 -1390.254} C_VEL
LIN {X 0,Y 587.315,Z 306.323,A -85,B 0,C 180,E1 -1393.006,E2 -1393.006} C_VEL
LIN {X 0,Y 587.316,Z 306.326,A -85,B 0,C 180,E1 -1395.887,E2 -1395.887} C_VEL
LIN {X 0,Y 587.327,Z 306.329,A -85,B 0,C 180,E1 -1398.925,E2 -1398.925} C_VEL
LIN {X 0,Y 587.314,Z 306.324,A -85,B 0,C 180,E1 -1401.519,E2 -1401.519} C_VEL
LIN {X 0,Y 587.344,Z 306.327,A -85,B 0,C 180,E1 -1404.103,E2 -1404.103} C_VEL
LIN {X 0,Y 587.338,Z 306.321,A -85,B 0,C 180,E1 -1406.887,E2 -1406.887} C_VEL
LIN {X 0,Y 587.323,Z 306.326,A -85,B 0,C 180,E1 -1409.491,E2 -1409.491} C_VEL
LIN {X 0,Y 587.284,Z 306.329,A -85,B 0,C 180,E1 -1412.179,E2 -1412.179} C_VEL
LIN {X 0,Y 587.326,Z 306.328,A -85,B 0,C 180,E1 -1414.483,E2 -1414.483} C_VEL
LIN {X 0,Y 587.337,Z 306.324,A -85,B 0,C 180,E1 -1417.486,E2 -1417.486} C_VEL
LIN {X 0,Y 587.329,Z 306.327,A -85,B 0,C 180,E1 -1419.695,E2 -1419.695} C_VEL
LIN {X 0,Y 587.339,Z 306.323,A -85,B 0,C 180,E1 -1422.594,E2 -1422.594} C_VEL
LIN {X 0,Y 587.324,Z 306.323,A -85,B 0,C 180,E1 -1425.753,E2 -1425.753} C_VEL
LIN {X 0,Y 587.342,Z 306.32,A -85,B 0,C 180,E1 -1428.866,E2 -1428.866} C_VEL
LIN {X 0,Y 587.367,Z 306.321,A -85,B 0,C 180,E1 -1431.745,E2 -1431.745} C_VEL
LIN {X 0,Y 587.366,Z 306.319,A -85,B 0,C 180,E1 -1434.507,E2 -1434.507} C_VEL
LIN {X 0,Y 587.353,Z 306.319,A -85,B 0,C 180,E1 -1437.257,E2 -1437.257} C_VEL
LIN {X 0,Y 587.376,Z 306.323,A -85,B 0,C 180,E1 -1440,E2 -1440} C_VEL
LIN {X 0,Y 587.349,Z 306.32,A -85,B 0,C 180,E1 -1442.743,E2 -1442.743} C_VEL
LIN {X 0,Y 587.367,Z 306.32,A -85,B 0,C 180,E1 -1445.493,E2 -1445.493} C_VEL
LIN {X 0,Y 587.369,Z 306.32,A -85,B 0,C 180,E1 -1448.255,E2 -1448.255} C_VEL
LIN {X 0,Y 587.342,Z 306.32,A -85,B 0,C 180,E1 -1451.134,E2 -1451.134} C_VEL
LIN {X 0,Y 587.311,Z 306.325,A -85,B 0,C 180,E1 -1454.242,E2 -1454.242} C_VEL
LIN {X 0,Y 587.338,Z 306.325,A -85,B 0,C 180,E1 -1457.406,E2 -1457.406} C_VEL
LIN {X 0,Y 587.328,Z 306.326,A -85,B 0,C 180,E1 -1460.305,E2 -1460.305} C_VEL
LIN {X 0,Y 587.319,Z 306.323,A -85,B 0,C 180,E1 -1463.259,E2 -1463.259} C_VEL
LIN {X 0,Y 587.329,Z 306.326,A -85,B 0,C 180,E1 -1465.517,E2 -1465.517} C_VEL
LIN {X 0,Y 587.283,Z 306.33,A -85,B 0,C 180,E1 -1467.821,E2 -1467.821} C_VEL
LIN {X 0,Y 587.322,Z 306.325,A -85,B 0,C 180,E1 -1470.509,E2 -1470.509} C_VEL
LIN {X 0,Y 587.336,Z 306.322,A -85,B 0,C 180,E1 -1473.112,E2 -1473.112} C_VEL
LIN {X 0,Y 587.344,Z 306.326,A -85,B 0,C 180,E1 -1475.896,E2 -1475.896} C_VEL
LIN {X 0,Y 587.317,Z 306.323,A -85,B 0,C 180,E1 -1478.481,E2 -1478.481} C_VEL
LIN {X 0,Y 587.327,Z 306.33,A -85,B 0,C 180,E1 -1481.158,E2 -1481.158} C_VEL
LIN {X 0,Y 587.3,Z 306.327,A -85,B 0,C 180,E1 -1484.111,E2 -1484.111} C_VEL
LIN {X 0,Y 587.313,Z 306.324,A -85,B 0,C 180,E1 -1486.994,E2 -1486.994} C_VEL
LIN {X 0,Y 587.313,Z 306.331,A -85,B 0,C 180,E1 -1489.746,E2 -1489.746} C_VEL
LIN {X 0,Y 587.34,Z 306.322,A -85,B 0,C 180,E1 -1492.392,E2 -1492.392} C_VEL
LIN {X 0,Y 587.338,Z 306.44,A -85,B 0,C 180,E1 -1493.998,E2 -1493.998} C_VEL
LIN {X 0,Y 587.483,Z 310.754,A -85,B 0,C 180,E1 -1495.633,E2 -1495.633} C_VEL
LIN {X 0,Y 587.457,Z 315.622,A -85,B 0,C 180,E1 -1497.429,E2 -1497.429} C_VEL
LIN {X 0,Y 587.463,Z 323.414,A -85,B 0,C 180,E1 -1500.233,E2 -1500.233} C_VEL
LIN {X 0,Y 587.385,Z 331.205,A -85,B 0,C 180,E1 -1502.957,E2 -1502.957} C_VEL
LIN {X 0,Y 587.356,Z 338.408,A -85,B 0,C 180,E1 -1505.42,E2 -1505.42} C_VEL
LIN {X 0,Y 587.342,Z 347.9,A -85,B 0,C 180,E1 -1508.595,E2 -1508.595} C_VEL
LIN {X 0,Y 587.272,Z 356.805,A -85,B 0,C 180,E1 -1511.511,E2 -1511.511} C_VEL
LIN {X 0,Y 587.245,Z 365.709,A -85,B 0,C 180,E1 -1514.379,E2 -1514.379} C_VEL
LIN {X 0,Y 587.201,Z 374.613,A -85,B 0,C 180,E1 -1517.208,E2 -1517.208} C_VEL
LIN {X 0,Y 587.173,Z 376.491,A -85,B 0,C 180,E1 -1517.8,E2 -1517.8} C_VEL
LIN {X 0,Y 587.747,Z 381.226,A -85,B 0,C 180,E1 -1517.899,E2 -1517.899} C_VEL
LIN {X 0,Y 587.679,Z 394.493,A -85,B 0,C 180,E1 -1518.226,E2 -1518.226} C_VEL
LIN {X 0,Y 587.564,Z 406.449,A -85,B 0,C 180,E1 -1518.658,E2 -1518.658} C_VEL
LIN {X 0,Y 587.476,Z 418.207,A -85,B 0,C 180,E1 -1519.227,E2 -1519.227} C_VEL
LIN {X 0,Y 587.462,Z 429.475,A -85,B 0,C 180,E1 -1519.923,E2 -1519.923} C_VEL
LIN {X 0,Y 587.384,Z 439.645,A -85,B 0,C 180,E1 -1520.704,E2 -1520.704} C_VEL
LIN {X 0,Y 587.34,Z 448.786,A -85,B 0,C 180,E1 -1521.571,E2 -1521.571} C_VEL
LIN {X 0,Y 587.259,Z 457.69,A -85,B 0,C 180,E1 -1522.608,E2 -1522.608} C_VEL
LIN {X 0,Y 587.195,Z 464.745,A -85,B 0,C 180,E1 -1523.627,E2 -1523.627} C_VEL
LIN {X 0,Y 587.211,Z 469.679,A -85,B 0,C 180,E1 -1524.505,E2 -1524.505} C_VEL
LIN {X 0,Y 587.188,Z 474.37,A -85,B 0,C 180,E1 -1525.538,E2 -1525.538} C_VEL
LIN {X 0,Y 587.193,Z 477.955,A -85,B 0,C 180,E1 -1526.569,E2 -1526.569} C_VEL
LIN {X 0,Y 587.132,Z 479.808,A -85,B 0,C 180,E1 -1527.255,E2 -1527.255} C_VEL
LIN {X 0,Y 587.141,Z 481.201,A -85,B 0,C 180,E1 -1527.942,E2 -1527.942} C_VEL
LIN {X 0,Y 587.14,Z 482.784,A -85,B 0,C 180,E1 -1529.314,E2 -1529.314} C_VEL
LIN {X 0,Y 587.137,Z 483,A -85,B 0,C 180,E1 -1530,E2 -1530} C_VEL
LIN {X 0,Y 587.147,Z 482.185,A -85,B 0,C 180,E1 -1531.371,E2 -1531.371} C_VEL
LIN {X 0,Y 587.141,Z 481.203,A -85,B 0,C 180,E1 -1532.058,E2 -1532.058} C_VEL
LIN {X 0,Y 587.132,Z 479.81,A -85,B 0,C 180,E1 -1532.744,E2 -1532.744} C_VEL
LIN {X 0,Y 587.213,Z 476.897,A -85,B 0,C 180,E1 -1533.774,E2 -1533.774} C_VEL
LIN {X 0,Y 587.147,Z 472.951,A -85,B 0,C 180,E1 -1534.806,E2 -1534.806} C_VEL
LIN {X 0,Y 587.218,Z 466.88,A -85,B 0,C 180,E1 -1536.011,E2 -1536.011} C_VEL
LIN {X 0,Y 587.244,Z 460.239,A -85,B 0,C 180,E1 -1537.046,E2 -1537.046} C_VEL
LIN {X 0,Y 587.299,Z 451.993,A -85,B 0,C 180,E1 -1538.083,E2 -1538.083} C_VEL
LIN {X 0,Y 587.343,Z 443.542,A -85,B 0,C 180,E1 -1538.948,E2 -1538.948} C_VEL
LIN {X 0,Y 587.416,Z 433.099,A -85,B 0,C 180,E1 -1539.816,E2 -1539.816} C_VEL
LIN {X 0,Y 587.471,Z 422.766,A -85,B 0,C 180,E1 -1540.511,E2 -1540.511} C_VEL
LIN {X 0,Y 587.529,Z 411.172,A -85,B 0,C 180,E1 -1541.133,E2 -1541.133} C_VEL
LIN {X 0,Y 587.606,Z 398.708,A -85,B 0,C 180,E1 -1541.636,E2 -1541.636} C_VEL
LIN {X 0,Y 587.745,Z 385.46,A -85,B 0,C 180,E1 -1542.013,E2 -1542.013} C_VEL
LIN {X 0,Y 587.528,Z 378.68,A -85,B 0,C 180,E1 -1542.154,E2 -1542.154} C_VEL
LIN {X 0,Y 587.173,Z 376.424,A -85,B 0,C 180,E1 -1542.222,E2 -1542.222} C_VEL
LIN {X 0,Y 587.216,Z 367.937,A -85,B 0,C 180,E1 -1544.91,E2 -1544.91} C_VEL
LIN {X 0,Y 587.282,Z 359.033,A -85,B 0,C 180,E1 -1547.767,E2 -1547.767} C_VEL
LIN {X 0,Y 587.298,Z 350.144,A -85,B 0,C 180,E1 -1550.666,E2 -1550.666} C_VEL
LIN {X 0,Y 587.345,Z 341.224,A -85,B 0,C 180,E1 -1553.631,E2 -1553.631} C_VEL
LIN {X 0,Y 587.366,Z 333.433,A -85,B 0,C 180,E1 -1556.276,E2 -1556.276} C_VEL
LIN {X 0,Y 587.467,Z 324.529,A -85,B 0,C 180,E1 -1559.372,E2 -1559.372} C_VEL
LIN {X 0,Y 587.459,Z 317.595,A -85,B 0,C 180,E1 -1561.853,E2 -1561.853} C_VEL
LIN {X 0,Y 587.481,Z 311.172,A -85,B 0,C 180,E1 -1564.211,E2 -1564.211} C_VEL
LIN {X 0,Y 587.337,Z 306.442,A -85,B 0,C 180,E1 -1566.002,E2 -1566.002} C_VEL
LIN {X 0,Y 587.325,Z 306.329,A -85,B 0,C 180,E1 -1568.478,E2 -1568.478} C_VEL
LIN {X 0,Y 587.334,Z 306.322,A -85,B 0,C 180,E1 -1571.156,E2 -1571.156} C_VEL
LIN {X 0,Y 587.329,Z 306.324,A -85,B 0,C 180,E1 -1574.113,E2 -1574.113} C_VEL
LIN {X 0,Y 587.293,Z 306.332,A -85,B 0,C 180,E1 -1576.991,E2 -1576.991} C_VEL
LIN {X 0,Y 587.3,Z 306.325,A -85,B 0,C 180,E1 -1579.744,E2 -1579.744} C_VEL
LIN {X 0,Y 587.337,Z 306.327,A -85,B 0,C 180,E1 -1582.392,E2 -1582.392} C_VEL
LIN {X 0,Y 587.342,Z 306.32,A -85,B 0,C 180,E1 -1584.945,E2 -1584.945} C_VEL
LIN {X 0,Y 587.334,Z 306.328,A -85,B 0,C 180,E1 -1587.421,E2 -1587.421} C_VEL
LIN {X 0,Y 587.304,Z 306.325,A -85,B 0,C 180,E1 -1589.828,E2 -1589.828} C_VEL
LIN {X 0,Y 587.286,Z 306.331,A -85,B 0,C 180,E1 -1592.317,E2 -1592.317} C_VEL
LIN {X 0,Y 587.342,Z 306.32,A -85,B 0,C 180,E1 -1595.241,E2 -1595.241} C_VEL
LIN {X 0,Y 587.319,Z 306.324,A -85,B 0,C 180,E1 -1598.226,E2 -1598.226} C_VEL
LIN {X 0,Y 587.341,Z 306.327,A -85,B 0,C 180,E1 -1601.151,E2 -1601.151} C_VEL
LIN {X 0,Y 587.311,Z 306.326,A -85,B 0,C 180,E1 -1603.31,E2 -1603.31} C_VEL
LIN {X 0,Y 587.338,Z 306.326,A -85,B 0,C 180,E1 -1606.154,E2 -1606.154} C_VEL
LIN {X 0,Y 587.324,Z 306.322,A -85,B 0,C 180,E1 -1608.962,E2 -1608.962} C_VEL
LIN {X 0,Y 587.365,Z 306.321,A -85,B 0,C 180,E1 -1611.745,E2 -1611.745} C_VEL
LIN {X 0,Y 587.366,Z 306.32,A -85,B 0,C 180,E1 -1614.507,E2 -1614.507} C_VEL
LIN {X 0,Y 587.349,Z 306.32,A -85,B 0,C 180,E1 -1617.257,E2 -1617.257} C_VEL
LIN {X 0,Y 587.372,Z 306.324,A -85,B 0,C 180,E1 -1620,E2 -1620} C_VEL
LIN {X 0,Y 587.349,Z 306.319,A -85,B 0,C 180,E1 -1622.743,E2 -1622.743} C_VEL
LIN {X 0,Y 587.365,Z 306.32,A -85,B 0,C 180,E1 -1625.493,E2 -1625.493} C_VEL
LIN {X 0,Y 587.365,Z 306.321,A -85,B 0,C 180,E1 -1628.255,E2 -1628.255} C_VEL
LIN {X 0,Y 587.336,Z 306.321,A -85,B 0,C 180,E1 -1631.134,E2 -1631.134} C_VEL
LIN {X 0,Y 587.326,Z 306.323,A -85,B 0,C 180,E1 -1634.25,E2 -1634.25} C_VEL
LIN {X 0,Y 587.342,Z 306.324,A -85,B 0,C 180,E1 -1637.406,E2 -1637.406} C_VEL
LIN {X 0,Y 587.314,Z 306.324,A -85,B 0,C 180,E1 -1638.32,E2 -1638.32} C_VEL
LIN {X 0,Y 586.662,Z 306.412,A -85,B 0,C 180,E1 -1638.892,E2 -1638.892} C_VEL
LIN {X 0,Y 583.834,Z 306.762,A -85,B 0,C 180,E1 -1639.821,E2 -1639.821} C_VEL
LIN {X 0,Y 581.426,Z 307.064,A -85,B 0,C 180,E1 -1640.568,E2 -1640.568} C_VEL
LIN {X 0,Y 580.374,Z 307.19,A -85,B 0,C 180,E1 -1641.144,E2 -1641.144} C_VEL
LIN {X 0,Y 580.279,Z 307.2,A -85,B 0,C 180,E1 -1641.339,E2 -1641.339} C_VEL
LIN {X 0,Y 580.293,Z 307.202,A -85,B 0,C 180,E1 -1644.317,E2 -1644.317} C_VEL
LIN {X 0,Y 580.257,Z 307.203,A -85,B 0,C 180,E1 -1646.625,E2 -1646.625} C_VEL
LIN {X 0,Y 580.255,Z 307.203,A -85,B 0,C 180,E1 -1649.775,E2 -1649.775} C_VEL
LIN {X 0,Y 580.295,Z 307.2,A -85,B 0,C 180,E1 -1652.201,E2 -1652.201} C_VEL
LIN {X 0,Y 580.293,Z 307.2,A -85,B 0,C 180,E1 -1654.696,E2 -1654.696} C_VEL
LIN {X 0,Y 580.293,Z 307.201,A -85,B 0,C 180,E1 -1657.269,E2 -1657.269} C_VEL
LIN {X 0,Y 580.28,Z 307.2,A -85,B 0,C 180,E1 -1660.271,E2 -1660.271} C_VEL
LIN {X 0,Y 580.234,Z 307.206,A -85,B 0,C 180,E1 -1663.388,E2 -1663.388} C_VEL
LIN {X 0,Y 580.274,Z 307.207,A -85,B 0,C 180,E1 -1666.343,E2 -1666.343} C_VEL
LIN {X 0,Y 580.297,Z 307.199,A -85,B 0,C 180,E1 -1669.158,E2 -1669.158} C_VEL
LIN {X 0,Y 580.284,Z 307.201,A -85,B 0,C 180,E1 -1671.928,E2 -1671.928} C_VEL
LIN {X 0,Y 580.206,Z 307.212,A -85,B 0,C 180,E1 -1674.451,E2 -1674.451} C_VEL
LIN {X 0,Y 580.282,Z 308.458,A -85,B 0,C 180,E1 -1675.444,E2 -1675.444} C_VEL
LIN {X 0,Y 580.25,Z 312.629,A -85,B 0,C 180,E1 -1677.978,E2 -1677.978} C_VEL
LIN {X 0,Y 580.18,Z 317.216,A -85,B 0,C 180,E1 -1680.712,E2 -1680.712} C_VEL
LIN {X 0,Y 580.169,Z 321.79,A -85,B 0,C 180,E1 -1683.372,E2 -1683.372} C_VEL
LIN {X 0,Y 580.14,Z 325.811,A -85,B 0,C 180,E1 -1685.677,E2 -1685.677} C_VEL
LIN {X 0,Y 580.126,Z 329.954,A -85,B 0,C 180,E1 -1687.942,E2 -1687.942} C_VEL
LIN {X 0,Y 580.135,Z 335.483,A -85,B 0,C 180,E1 -1690.909,E2 -1690.909} C_VEL
LIN {X 0,Y 580.086,Z 341.013,A -85,B 0,C 180,E1 -1693.821,E2 -1693.821} C_VEL
LIN {X 0,Y 580.095,Z 345.16,A -85,B 0,C 180,E1 -1695.978,E2 -1695.978} C_VEL
LIN {X 0,Y 580.07,Z 348.53,A -85,B 0,C 180,E1 -1697.715,E2 -1697.715} C_VEL
LIN {X 0,Y 580.789,Z 354.515,A -85,B 0,C 180,E1 -1697.863,E2 -1697.863} C_VEL
LIN {X 0,Y 580.679,Z 367.17,A -85,B 0,C 180,E1 -1698.216,E2 -1698.216} C_VEL
LIN {X 0,Y 580.577,Z 378.891,A -85,B 0,C 180,E1 -1698.674,E2 -1698.674} C_VEL
LIN {X 0,Y 580.499,Z 390.558,A -85,B 0,C 180,E1 -1699.273,E2 -1699.273} C_VEL
LIN {X 0,Y 580.448,Z 401.334,A -85,B 0,C 180,E1 -1699.977,E2 -1699.977} C_VEL
LIN {X 0,Y 580.333,Z 411.108,A -85,B 0,C 180,E1 -1700.767,E2 -1700.767} C_VEL
LIN {X 0,Y 580.264,Z 420,A -85,B 0,C 180,E1 -1701.643,E2 -1701.643} C_VEL
LIN {X 0,Y 580.205,Z 428.683,A -85,B 0,C 180,E1 -1702.693,E2 -1702.693} C_VEL
LIN {X 0,Y 580.137,Z 435.61,A -85,B 0,C 180,E1 -1703.741,E2 -1703.741} C_VEL
LIN {X 0,Y 580.085,Z 441.159,A -85,B 0,C 180,E1 -1704.787,E2 -1704.787} C_VEL
LIN {X 0,Y 580.105,Z 445.519,A -85,B 0,C 180,E1 -1705.832,E2 -1705.832} C_VEL
LIN {X 0,Y 580.123,Z 447.822,A -85,B 0,C 180,E1 -1706.528,E2 -1706.528} C_VEL
LIN {X 0,Y 580.043,Z 449.699,A -85,B 0,C 180,E1 -1707.222,E2 -1707.222} C_VEL
LIN {X 0,Y 580.04,Z 451.128,A -85,B 0,C 180,E1 -1707.917,E2 -1707.917} C_VEL
LIN {X 0,Y 580.04,Z 452.755,A -85,B 0,C 180,E1 -1709.306,E2 -1709.306} C_VEL
LIN {X 0,Y 580.038,Z 452.996,A -85,B 0,C 180,E1 -1710,E2 -1710} C_VEL
LIN {X 0,Y 580.04,Z 452.815,A -85,B 0,C 180,E1 -1710.695,E2 -1710.695} C_VEL
LIN {X 0,Y 580.04,Z 451.272,A -85,B 0,C 180,E1 -1712.083,E2 -1712.083} C_VEL
LIN {X 0,Y 580.044,Z 449.91,A -85,B 0,C 180,E1 -1712.778,E2 -1712.778} C_VEL
LIN {X 0,Y 580.11,Z 447.033,A -85,B 0,C 180,E1 -1713.821,E2 -1713.821} C_VEL
LIN {X 0,Y 580.053,Z 443.133,A -85,B 0,C 180,E1 -1714.865,E2 -1714.865} C_VEL
LIN {X 0,Y 580.163,Z 438.101,A -85,B 0,C 180,E1 -1715.91,E2 -1715.91} C_VEL
LIN {X 0,Y 580.158,Z 431.779,A -85,B 0,C 180,E1 -1716.958,E2 -1716.958} C_VEL
LIN {X 0,Y 580.241,Z 423.859,A -85,B 0,C 180,E1 -1718.007,E2 -1718.007} C_VEL
LIN {X 0,Y 580.308,Z 414.01,A -85,B 0,C 180,E1 -1719.058,E2 -1719.058} C_VEL
LIN {X 0,Y 580.416,Z 403.689,A -85,B 0,C 180,E1 -1719.936,E2 -1719.936} C_VEL
LIN {X 0,Y 580.487,Z 392.055,A -85,B 0,C 180,E1 -1720.728,E2 -1720.728} C_VEL
LIN {X 0,Y 580.548,Z 381.21,A -85,B 0,C 180,E1 -1721.312,E2 -1721.312} C_VEL
LIN {X 0,Y 580.673,Z 368.622,A -85,B 0,C 180,E1 -1721.825,E2 -1721.825} C_VEL
LIN {X 0,Y 580.773,Z 355.463,A -85,B 0,C 180,E1 -1722.204,E2 -1722.204} C_VEL
LIN {X 0,Y 580.468,Z 351.257,A -85,B 0,C 180,E1 -1722.299,E2 -1722.299} C_VEL
LIN {X 0,Y 580.082,Z 348.531,A -85,B 0,C 180,E1 -1722.374,E2 -1722.374} C_VEL
LIN {X 0,Y 580.101,Z 343.95,A -85,B 0,C 180,E1 -1724.739,E2 -1724.739} C_VEL
LIN {X 0,Y 580.052,Z 338.418,A -85,B 0,C 180,E1 -1727.632,E2 -1727.632} C_VEL
LIN {X 0,Y 580.097,Z 334.268,A -85,B 0,C 180,E1 -1729.83,E2 -1729.83} C_VEL
LIN {X 0,Y 580.127,Z 330.119,A -85,B 0,C 180,E1 -1732.058,E2 -1732.058} C_VEL
LIN {X 0,Y 580.155,Z 324.63,A -85,B 0,C 180,E1 -1735.087,E2 -1735.087} C_VEL
LIN {X 0,Y 580.212,Z 319.84,A -85,B 0,C 180,E1 -1737.842,E2 -1737.842} C_VEL
LIN {X 0,Y 580.197,Z 315.03,A -85,B 0,C 180,E1 -1740.679,E2 -1740.679} C_VEL
LIN {X 0,Y 580.271,Z 310.644,A -85,B 0,C 180,E1 -1743.311,E2 -1743.311} C_VEL
LIN {X 0,Y 580.27,Z 308.375,A -85,B 0,C 180,E1 -1744.697,E2 -1744.697} C_VEL
LIN {X 0,Y 580.208,Z 307.212,A -85,B 0,C 180,E1 -1745.55,E2 -1745.55} C_VEL
LIN {X 0,Y 580.282,Z 307.201,A -85,B 0,C 180,E1 -1748.146,E2 -1748.146} C_VEL
LIN {X 0,Y 580.298,Z 307.199,A -85,B 0,C 180,E1 -1750.843,E2 -1750.843} C_VEL
LIN {X 0,Y 580.279,Z 307.205,A -85,B 0,C 180,E1 -1753.657,E2 -1753.657} C_VEL
LIN {X 0,Y 580.238,Z 307.205,A -85,B 0,C 180,E1 -1756.613,E2 -1756.613} C_VEL
LIN {X 0,Y 580.289,Z 307.204,A -85,B 0,C 180,E1 -1759.156,E2 -1759.156} C_VEL
LIN {X 0,Y 580.282,Z 307.202,A -85,B 0,C 180,E1 -1761.927,E2 -1761.927} C_VEL
LIN {X 0,Y 580.284,Z 307.202,A -85,B 0,C 180,E1 -1764.455,E2 -1764.455} C_VEL
LIN {X 0,Y 580.29,Z 307.2,A -85,B 0,C 180,E1 -1766.975,E2 -1766.975} C_VEL
LIN {X 0,Y 580.285,Z 307.203,A -85,B 0,C 180,E1 -1769.424,E2 -1769.424} C_VEL
LIN {X 0,Y 580.238,Z 307.206,A -85,B 0,C 180,E1 -1772.151,E2 -1772.151} C_VEL
LIN {X 0,Y 580.283,Z 307.201,A -85,B 0,C 180,E1 -1774.919,E2 -1774.919} C_VEL
LIN {X 0,Y 580.272,Z 307.206,A -85,B 0,C 180,E1 -1777.947,E2 -1777.947} C_VEL
LIN {X 0,Y 580.314,Z 307.199,A -85,B 0,C 180,E1 -1780.914,E2 -1780.914} C_VEL
LIN {X 0,Y 580.257,Z 307.202,A -85,B 0,C 180,E1 -1783.825,E2 -1783.825} C_VEL
LIN {X 0,Y 580.296,Z 307.2,A -85,B 0,C 180,E1 -1785.982,E2 -1785.982} C_VEL
LIN {X 0,Y 580.299,Z 307.198,A -85,B 0,C 180,E1 -1788.827,E2 -1788.827} C_VEL
LIN {X 0,Y 580.33,Z 307.199,A -85,B 0,C 180,E1 -1791.644,E2 -1791.644} C_VEL
LIN {X 0,Y 580.332,Z 307.195,A -85,B 0,C 180,E1 -1794.44,E2 -1794.44} C_VEL
LIN {X 0,Y 580.322,Z 307.195,A -85,B 0,C 180,E1 -1797.223,E2 -1797.223} C_VEL
LIN {X 0,Y 580.345,Z 307.198,A -85,B 0,C 180,E1 -1800,E2 -1800} C_VEL
LIN {X 0,Y 580.318,Z 307.196,A -85,B 0,C 180,E1 -1802.777,E2 -1802.777} C_VEL
LIN {X 0,Y 580.334,Z 307.196,A -85,B 0,C 180,E1 -1805.56,E2 -1805.56} C_VEL
LIN {X 0,Y 580.332,Z 307.198,A -85,B 0,C 180,E1 -1808.356,E2 -1808.356} C_VEL
LIN {X 0,Y 580.294,Z 307.198,A -85,B 0,C 180,E1 -1811.191,E2 -1811.191} C_VEL
LIN {X 0,Y 580.287,Z 307.203,A -85,B 0,C 180,E1 -1814.018,E2 -1814.018} C_VEL
LIN {X 0,Y 580.307,Z 307.201,A -85,B 0,C 180,E1 -1816.914,E2 -1816.914} C_VEL
LIN {X 0,Y 580.302,Z 307.197,A -85,B 0,C 180,E1 -1819.822,E2 -1819.822} C_VEL
LIN {X 0,Y 580.272,Z 307.205,A -85,B 0,C 180,E1 -1822.053,E2 -1822.053} C_VEL
LIN {X 0,Y 580.302,Z 307.197,A -85,B 0,C 180,E1 -1825.08,E2 -1825.08} C_VEL
LIN {X 0,Y 580.23,Z 307.206,A -85,B 0,C 180,E1 -1828.189,E2 -1828.189} C_VEL
LIN {X 0,Y 580.276,Z 307.206,A -85,B 0,C 180,E1 -1830.694,E2 -1830.694} C_VEL
LIN {X 0,Y 580.3,Z 307.198,A -85,B 0,C 180,E1 -1833.317,E2 -1833.317} C_VEL
LIN {X 0,Y 580.29,Z 307.201,A -85,B 0,C 180,E1 -1836.402,E2 -1836.402} C_VEL
LIN {X 0,Y 580.286,Z 307.203,A -85,B 0,C 180,E1 -1839.185,E2 -1839.185} C_VEL
LIN {X 0,Y 580.246,Z 307.204,A -85,B 0,C 180,E1 -1841.772,E2 -1841.772} C_VEL
LIN {X 0,Y 580.25,Z 307.211,A -85,B 0,C 180,E1 -1844.628,E2 -1844.628} C_VEL
LIN {X 0,Y 580.285,Z 307.202,A -85,B 0,C 180,E1 -1847.629,E2 -1847.629} C_VEL
LIN {X 0,Y 580.283,Z 307.203,A -85,B 0,C 180,E1 -1850.067,E2 -1850.067} C_VEL
LIN {X 0,Y 580.277,Z 307.208,A -85,B 0,C 180,E1 -1853.069,E2 -1853.069} C_VEL
LIN {X 0,Y 580.304,Z 307.38,A -85,B 0,C 180,E1 -1853.855,E2 -1853.855} C_VEL
LIN {X 0,Y 580.516,Z 311.17,A -85,B 0,C 180,E1 -1855.32,E2 -1855.32} C_VEL
LIN {X 0,Y 580.47,Z 318.209,A -85,B 0,C 180,E1 -1857.943,E2 -1857.943} C_VEL
LIN {X 0,Y 580.453,Z 325.719,A -85,B 0,C 180,E1 -1860.664,E2 -1860.664} C_VEL
LIN {X 0,Y 580.351,Z 334.219,A -85,B 0,C 180,E1 -1863.655,E2 -1863.655} C_VEL
LIN {X 0,Y 580.302,Z 342.335,A -85,B 0,C 180,E1 -1866.443,E2 -1866.443} C_VEL
LIN {X 0,Y 580.264,Z 349.464,A -85,B 0,C 180,E1 -1868.845,E2 -1868.845} C_VEL
LIN {X 0,Y 580.198,Z 357.918,A -85,B 0,C 180,E1 -1871.643,E2 -1871.643} C_VEL
LIN {X 0,Y 580.175,Z 366.822,A -85,B 0,C 180,E1 -1874.544,E2 -1874.544} C_VEL
LIN {X 0,Y 580.129,Z 375.726,A -85,B 0,C 180,E1 -1877.405,E2 -1877.405} C_VEL
LIN {X 0,Y 580.104,Z 376.491,A -85,B 0,C 180,E1 -1877.649,E2 -1877.649} C_VEL
LIN {X 0,Y 580.806,Z 382.368,A -85,B 0,C 180,E1 -1877.775,E2 -1877.775} C_VEL
LIN {X 0,Y 580.731,Z 394.494,A -85,B 0,C 180,E1 -1878.083,E2 -1878.083} C_VEL
LIN {X 0,Y 580.615,Z 406.319,A -85,B 0,C 180,E1 -1878.515,E2 -1878.515} C_VEL
LIN {X 0,Y 580.485,Z 418.207,A -85,B 0,C 180,E1 -1879.095,E2 -1879.095} C_VEL
LIN {X 0,Y 580.451,Z 429.475,A -85,B 0,C 180,E1 -1879.8,E2 -1879.8} C_VEL
LIN {X 0,Y 580.352,Z 439.645,A -85,B 0,C 180,E1 -1880.591,E2 -1880.591} C_VEL
LIN {X 0,Y 580.279,Z 448.786,A -85,B 0,C 180,E1 -1881.468,E2 -1881.468} C_VEL
LIN {X 0,Y 580.199,Z 457.69,A -85,B 0,C 180,E1 -1882.518,E2 -1882.518} C_VEL
LIN {X 0,Y 580.12,Z 464.465,A -85,B 0,C 180,E1 -1883.505,E2 -1883.505} C_VEL
LIN {X 0,Y 580.139,Z 469.679,A -85,B 0,C 180,E1 -1884.438,E2 -1884.438} C_VEL
LIN {X 0,Y 580.108,Z 474.37,A -85,B 0,C 180,E1 -1885.483,E2 -1885.483} C_VEL
LIN {X 0,Y 580.123,Z 477.956,A -85,B 0,C 180,E1 -1886.527,E2 -1886.527} C_VEL
LIN {X 0,Y 580.043,Z 479.808,A -85,B 0,C 180,E1 -1887.222,E2 -1887.222} C_VEL
LIN {X 0,Y 580.04,Z 481.201,A -85,B 0,C 180,E1 -1887.917,E2 -1887.917} C_VEL
LIN {X 0,Y 580.04,Z 482.784,A -85,B 0,C 180,E1 -1889.305,E2 -1889.305} C_VEL
LIN {X 0,Y 580.037,Z 483,A -85,B 0,C 180,E1 -1890,E2 -1890} C_VEL
LIN {X 0,Y 580.047,Z 482.185,A -85,B 0,C 180,E1 -1891.388,E2 -1891.388} C_VEL
LIN {X 0,Y 580.04,Z 481.202,A -85,B 0,C 180,E1 -1892.083,E2 -1892.083} C_VEL
LIN {X 0,Y 580.043,Z 479.81,A -85,B 0,C 180,E1 -1892.778,E2 -1892.778} C_VEL
LIN {X 0,Y 580.11,Z 476.897,A -85,B 0,C 180,E1 -1893.82,E2 -1893.82} C_VEL
LIN {X 0,Y 580.053,Z 472.951,A -85,B 0,C 180,E1 -1894.865,E2 -1894.865} C_VEL
LIN {X 0,Y 580.139,Z 466.88,A -85,B 0,C 180,E1 -1896.084,E2 -1896.084} C_VEL
LIN {X 0,Y 580.184,Z 460.239,A -85,B 0,C 180,E1 -1897.132,E2 -1897.132} C_VEL
LIN {X 0,Y 580.25,Z 451.994,A -85,B 0,C 180,E1 -1898.181,E2 -1898.181} C_VEL
LIN {X 0,Y 580.308,Z 443.542,A -85,B 0,C 180,E1 -1899.058,E2 -1899.058} C_VEL
LIN {X 0,Y 580.417,Z 433.1,A -85,B 0,C 180,E1 -1899.935,E2 -1899.935} C_VEL
LIN {X 0,Y 580.474,Z 422.767,A -85,B 0,C 180,E1 -1900.639,E2 -1900.639} C_VEL
LIN {X 0,Y 580.562,Z 411.604,A -85,B 0,C 180,E1 -1901.247,E2 -1901.247} C_VEL
LIN {X 0,Y 580.63,Z 399.783,A -85,B 0,C 180,E1 -1901.741,E2 -1901.741} C_VEL
LIN {X 0,Y 580.778,Z 386.374,A -85,B 0,C 180,E1 -1902.137,E2 -1902.137} C_VEL
LIN {X 0,Y 580.612,Z 379.689,A -85,B 0,C 180,E1 -1902.282,E2 -1902.282} C_VEL
LIN {X 0,Y 580.104,Z 376.493,A -85,B 0,C 180,E1 -1902.351,E2 -1902.351} C_VEL
LIN {X 0,Y 580.154,Z 367.937,A -85,B 0,C 180,E1 -1905.096,E2 -1905.096} C_VEL
LIN {X 0,Y 580.206,Z 359.033,A -85,B 0,C 180,E1 -1907.991,E2 -1907.991} C_VEL
LIN {X 0,Y 580.242,Z 351.241,A -85,B 0,C 180,E1 -1910.563,E2 -1910.563} C_VEL
LIN {X 0,Y 580.268,Z 343.973,A -85,B 0,C 180,E1 -1913.002,E2 -1913.002} C_VEL
LIN {X 0,Y 580.321,Z 335.659,A -85,B 0,C 180,E1 -1915.847,E2 -1915.847} C_VEL
LIN {X 0,Y 580.371,Z 327.868,A -85,B 0,C 180,E1 -1918.575,E2 -1918.575} C_VEL
LIN {X 0,Y 580.422,Z 321.887,A -85,B 0,C 180,E1 -1920.717,E2 -1920.717} C_VEL
LIN {X 0,Y 580.528,Z 314.708,A -85,B 0,C 180,E1 -1923.35,E2 -1923.35} C_VEL
LIN {X 0,Y 580.462,Z 308.283,A -85,B 0,C 180,E1 -1925.785,E2 -1925.785} C_VEL
LIN {X 0,Y 580.259,Z 307.209,A -85,B 0,C 180,E1 -1926.233,E2 -1926.233} C_VEL
LIN {X 0,Y 580.303,Z 307.199,A -85,B 0,C 180,E1 -1929.186,E2 -1929.186} C_VEL
LIN {X 0,Y 580.31,Z 307.201,A -85,B 0,C 180,E1 -1931.765,E2 -1931.765} C_VEL
LIN {X 0,Y 580.263,Z 307.202,A -85,B 0,C 180,E1 -1934.625,E2 -1934.625} C_VEL
LIN {X 0,Y 580.253,Z 307.209,A -85,B 0,C 180,E1 -1937.291,E2 -1937.291} C_VEL
LIN {X 0,Y 580.276,Z 307.201,A -85,B 0,C 180,E1 -1940.066,E2 -1940.066} C_VEL
LIN {X 0,Y 580.295,Z 307.198,A -85,B 0,C 180,E1 -1943.064,E2 -1943.064} C_VEL
LIN {X 0,Y 580.296,Z 307.202,A -85,B 0,C 180,E1 -1945.44,E2 -1945.44} C_VEL
LIN {X 0,Y 580.301,Z 307.199,A -85,B 0,C 180,E1 -1947.967,E2 -1947.967} C_VEL
LIN {X 0,Y 580.264,Z 307.207,A -85,B 0,C 180,E1 -1950.694,E2 -1950.694} C_VEL
LIN {X 0,Y 580.272,Z 307.201,A -85,B 0,C 180,E1 -1953.667,E2 -1953.667} C_VEL
LIN {X 0,Y 580.293,Z 307.201,A -85,B 0,C 180,E1 -1955.683,E2 -1955.683} C_VEL
LIN {X 0,Y 580.282,Z 307.2,A -85,B 0,C 180,E1 -1958.694,E2 -1958.694} C_VEL
LIN {X 0,Y 580.308,Z 307.201,A -85,B 0,C 180,E1 -1960.914,E2 -1960.914} C_VEL
LIN {X 0,Y 580.252,Z 307.204,A -85,B 0,C 180,E1 -1963.825,E2 -1963.825} C_VEL
LIN {X 0,Y 580.298,Z 307.201,A -85,B 0,C 180,E1 -1965.982,E2 -1965.982} C_VEL
LIN {X 0,Y 580.293,Z 307.198,A -85,B 0,C 180,E1 -1968.827,E2 -1968.827} C_VEL
LIN {X 0,Y 580.328,Z 307.199,A -85,B 0,C 180,E1 -1971.644,E2 -1971.644} C_VEL
LIN {X 0,Y 580.332,Z 307.196,A -85,B 0,C 180,E1 -1974.44,E2 -1974.44} C_VEL
LIN {X 0,Y 580.318,Z 307.196,A -85,B 0,C 180,E1 -1977.223,E2 -1977.223} C_VEL
LIN {X 0,Y 580.341,Z 307.199,A -85,B 0,C 180,E1 -1980,E2 -1980} C_VEL
LIN {X 0,Y 580.317,Z 307.195,A -85,B 0,C 180,E1 -1982.777,E2 -1982.777} C_VEL
LIN {X 0,Y 580.332,Z 307.196,A -85,B 0,C 180,E1 -1985.56,E2 -1985.56} C_VEL
LIN {X 0,Y 580.328,Z 307.199,A -85,B 0,C 180,E1 -1988.356,E2 -1988.356} C_VEL
LIN {X 0,Y 580.288,Z 307.199,A -85,B 0,C 180,E1 -1991.191,E2 -1991.191} C_VEL
LIN {X 0,Y 580.298,Z 307.201,A -85,B 0,C 180,E1 -1994.018,E2 -1994.018} C_VEL
LIN {X 0,Y 580.301,Z 307.201,A -85,B 0,C 180,E1 -1996.914,E2 -1996.914} C_VEL
LIN {X 0,Y 580.3,Z 307.198,A -85,B 0,C 180,E1 -1999.823,E2 -1999.823} C_VEL
LIN {X 0,Y 580.279,Z 307.2,A -85,B 0,C 180,E1 -2001.339,E2 -2001.339} C_VEL
LIN {X 0,Y 579.582,Z 307.291,A -85,B 0,C 180,E1 -2001.918,E2 -2001.918} C_VEL
LIN {X 0,Y 576.704,Z 307.647,A -85,B 0,C 180,E1 -2002.858,E2 -2002.858} C_VEL
LIN {X 0,Y 574.308,Z 307.947,A -85,B 0,C 180,E1 -2003.614,E2 -2003.614} C_VEL
LIN {X 0,Y 573.309,Z 308.073,A -85,B 0,C 180,E1 -2004.198,E2 -2004.198} C_VEL
LIN {X 0,Y 573.242,Z 308.078,A -85,B 0,C 180,E1 -2004.396,E2 -2004.396} C_VEL
LIN {X 0,Y 573.193,Z 308.085,A -85,B 0,C 180,E1 -2006.979,E2 -2006.979} C_VEL
LIN {X 0,Y 573.212,Z 308.083,A -85,B 0,C 180,E1 -2009.484,E2 -2009.484} C_VEL
LIN {X 0,Y 573.248,Z 308.078,A -85,B 0,C 180,E1 -2012.23,E2 -2012.23} C_VEL
LIN {X 0,Y 573.244,Z 308.078,A -85,B 0,C 180,E1 -2014.775,E2 -2014.775} C_VEL
LIN {X 0,Y 573.247,Z 308.078,A -85,B 0,C 180,E1 -2017.167,E2 -2017.167} C_VEL
LIN {X 0,Y 573.233,Z 308.083,A -85,B 0,C 180,E1 -2019.608,E2 -2019.608} C_VEL
LIN {X 0,Y 573.213,Z 308.085,A -85,B 0,C 180,E1 -2022.64,E2 -2022.64} C_VEL
LIN {X 0,Y 573.23,Z 308.078,A -85,B 0,C 180,E1 -2025.668,E2 -2025.668} C_VEL
LIN {X 0,Y 573.241,Z 308.078,A -85,B 0,C 180,E1 -2028.545,E2 -2028.545} C_VEL
LIN {X 0,Y 573.243,Z 308.083,A -85,B 0,C 180,E1 -2031.3,E2 -2031.3} C_VEL
LIN {X 0,Y 573.179,Z 308.085,A -85,B 0,C 180,E1 -2034.024,E2 -2034.024} C_VEL
LIN {X 0,Y 573.175,Z 308.304,A -85,B 0,C 180,E1 -2034.811,E2 -2034.811} C_VEL
LIN {X 0,Y 573.189,Z 312.439,A -85,B 0,C 180,E1 -2037.352,E2 -2037.352} C_VEL
LIN {X 0,Y 573.133,Z 316.496,A -85,B 0,C 180,E1 -2039.818,E2 -2039.818} C_VEL
LIN {X 0,Y 573.151,Z 320.542,A -85,B 0,C 180,E1 -2042.229,E2 -2042.229} C_VEL
LIN {X 0,Y 573.102,Z 325.575,A -85,B 0,C 180,E1 -2045.158,E2 -2045.158} C_VEL
LIN {X 0,Y 573.041,Z 329.955,A -85,B 0,C 180,E1 -2047.655,E2 -2047.655} C_VEL
LIN {X 0,Y 573.014,Z 334.102,A -85,B 0,C 180,E1 -2049.915,E2 -2049.915} C_VEL
LIN {X 0,Y 572.973,Z 338.249,A -85,B 0,C 180,E1 -2052.143,E2 -2052.143} C_VEL
LIN {X 0,Y 572.997,Z 343.779,A -85,B 0,C 180,E1 -2055.075,E2 -2055.075} C_VEL
LIN {X 0,Y 572.982,Z 348.531,A -85,B 0,C 180,E1 -2057.561,E2 -2057.561} C_VEL
LIN {X 0,Y 573.848,Z 354.537,A -85,B 0,C 180,E1 -2057.714,E2 -2057.714} C_VEL
LIN {X 0,Y 573.725,Z 367.185,A -85,B 0,C 180,E1 -2058.071,E2 -2058.071} C_VEL
LIN {X 0,Y 573.602,Z 379.878,A -85,B 0,C 180,E1 -2058.578,E2 -2058.578} C_VEL
LIN {X 0,Y 573.518,Z 390.792,A -85,B 0,C 180,E1 -2059.153,E2 -2059.153} C_VEL
LIN {X 0,Y 573.456,Z 401.34,A -85,B 0,C 180,E1 -2059.854,E2 -2059.854} C_VEL
LIN {X 0,Y 573.321,Z 411.114,A -85,B 0,C 180,E1 -2060.653,E2 -2060.653} C_VEL
LIN {X 0,Y 573.235,Z 420.005,A -85,B 0,C 180,E1 -2061.54,E2 -2061.54} C_VEL
LIN {X 0,Y 573.125,Z 428.688,A -85,B 0,C 180,E1 -2062.603,E2 -2062.603} C_VEL
LIN {X 0,Y 573.049,Z 435.613,A -85,B 0,C 180,E1 -2063.663,E2 -2063.663} C_VEL
LIN {X 0,Y 573.009,Z 441.161,A -85,B 0,C 180,E1 -2064.722,E2 -2064.722} C_VEL
LIN {X 0,Y 573.031,Z 445.521,A -85,B 0,C 180,E1 -2065.78,E2 -2065.78} C_VEL
LIN {X 0,Y 573.022,Z 447.825,A -85,B 0,C 180,E1 -2066.485,E2 -2066.485} C_VEL
LIN {X 0,Y 572.959,Z 449.701,A -85,B 0,C 180,E1 -2067.188,E2 -2067.188} C_VEL
LIN {X 0,Y 572.94,Z 451.128,A -85,B 0,C 180,E1 -2067.891,E2 -2067.891} C_VEL
LIN {X 0,Y 572.941,Z 452.755,A -85,B 0,C 180,E1 -2069.297,E2 -2069.297} C_VEL
LIN {X 0,Y 572.939,Z 452.996,A -85,B 0,C 180,E1 -2070,E2 -2070} C_VEL
LIN {X 0,Y 572.94,Z 452.814,A -85,B 0,C 180,E1 -2070.703,E2 -2070.703} C_VEL
LIN {X 0,Y 572.94,Z 451.27,A -85,B 0,C 180,E1 -2072.109,E2 -2072.109} C_VEL
LIN {X 0,Y 572.96,Z 449.909,A -85,B 0,C 180,E1 -2072.813,E2 -2072.813} C_VEL
LIN {X 0,Y 573.015,Z 447.031,A -85,B 0,C 180,E1 -2073.868,E2 -2073.868} C_VEL
LIN {X 0,Y 572.963,Z 443.131,A -85,B 0,C 180,E1 -2074.926,E2 -2074.926} C_VEL
LIN {X 0,Y 573.076,Z 438.098,A -85,B 0,C 180,E1 -2075.984,E2 -2075.984} C_VEL
LIN {X 0,Y 573.083,Z 431.775,A -85,B 0,C 180,E1 -2077.044,E2 -2077.044} C_VEL
LIN {X 0,Y 573.175,Z 423.854,A -85,B 0,C 180,E1 -2078.106,E2 -2078.106} C_VEL
LIN {X 0,Y 573.287,Z 414.004,A -85,B 0,C 180,E1 -2079.17,E2 -2079.17} C_VEL
LIN {X 0,Y 573.419,Z 403.683,A -85,B 0,C 180,E1 -2080.059,E2 -2080.059} C_VEL
LIN {X 0,Y 573.499,Z 392.26,A -85,B 0,C 180,E1 -2080.847,E2 -2080.847} C_VEL
LIN {X 0,Y 573.584,Z 381.198,A -85,B 0,C 180,E1 -2081.451,E2 -2081.451} C_VEL
LIN {X 0,Y 573.743,Z 368.607,A -85,B 0,C 180,E1 -2081.97,E2 -2081.97} C_VEL
LIN {X 0,Y 573.849,Z 355.439,A -85,B 0,C 180,E1 -2082.354,E2 -2082.354} C_VEL
LIN {X 0,Y 573.425,Z 351.511,A -85,B 0,C 180,E1 -2082.447,E2 -2082.447} C_VEL
LIN {X 0,Y 572.972,Z 348.53,A -85,B 0,C 180,E1 -2082.53,E2 -2082.53} C_VEL
LIN {X 0,Y 572.997,Z 343.949,A -85,B 0,C 180,E1 -2084.926,E2 -2084.926} C_VEL
LIN {X 0,Y 572.966,Z 338.417,A -85,B 0,C 180,E1 -2087.857,E2 -2087.857} C_VEL
LIN {X 0,Y 573.015,Z 334.267,A -85,B 0,C 180,E1 -2090.085,E2 -2090.085} C_VEL
LIN {X 0,Y 573.042,Z 330.118,A -85,B 0,C 180,E1 -2092.346,E2 -2092.346} C_VEL
LIN {X 0,Y 573.088,Z 324.74,A -85,B 0,C 180,E1 -2095.418,E2 -2095.418} C_VEL
LIN {X 0,Y 573.144,Z 320.296,A -85,B 0,C 180,E1 -2098.008,E2 -2098.008} C_VEL
LIN {X 0,Y 573.15,Z 315.298,A -85,B 0,C 180,E1 -2100.998,E2 -2100.998} C_VEL
LIN {X 0,Y 573.242,Z 311.152,A -85,B 0,C 180,E1 -2103.52,E2 -2103.52} C_VEL
LIN {X 0,Y 573.177,Z 308.449,A -85,B 0,C 180,E1 -2105.19,E2 -2105.19} C_VEL
LIN {X 0,Y 573.182,Z 308.084,A -85,B 0,C 180,E1 -2106.053,E2 -2106.053} C_VEL
LIN {X 0,Y 573.237,Z 308.085,A -85,B 0,C 180,E1 -2108.702,E2 -2108.702} C_VEL
LIN {X 0,Y 573.253,Z 308.077,A -85,B 0,C 180,E1 -2111.595,E2 -2111.595} C_VEL
LIN {X 0,Y 573.235,Z 308.078,A -85,B 0,C 180,E1 -2114.333,E2 -2114.333} C_VEL
LIN {X 0,Y 573.216,Z 308.086,A -85,B 0,C 180,E1 -2117.36,E2 -2117.36} C_VEL
LIN {X 0,Y 573.228,Z 308.082,A -85,B 0,C 180,E1 -2120.391,E2 -2120.391} C_VEL
LIN {X 0,Y 573.253,Z 308.076,A -85,B 0,C 180,E1 -2123.077,E2 -2123.077} C_VEL
LIN {X 0,Y 573.265,Z 308.08,A -85,B 0,C 180,E1 -2125.671,E2 -2125.671} C_VEL
LIN {X 0,Y 573.245,Z 308.076,A -85,B 0,C 180,E1 -2128.185,E2 -2128.185} C_VEL
LIN {X 0,Y 573.234,Z 308.08,A -85,B 0,C 180,E1 -2130.632,E2 -2130.632} C_VEL
LIN {X 0,Y 573.205,Z 308.081,A -85,B 0,C 180,E1 -2133.513,E2 -2133.513} C_VEL
LIN {X 0,Y 573.218,Z 308.086,A -85,B 0,C 180,E1 -2136.134,E2 -2136.134} C_VEL
LIN {X 0,Y 573.258,Z 308.078,A -85,B 0,C 180,E1 -2139.174,E2 -2139.174} C_VEL
LIN {X 0,Y 573.225,Z 308.083,A -85,B 0,C 180,E1 -2141.411,E2 -2141.411} C_VEL
LIN {X 0,Y 573.233,Z 308.077,A -85,B 0,C 180,E1 -2143.621,E2 -2143.621} C_VEL
LIN {X 0,Y 573.242,Z 308.078,A -85,B 0,C 180,E1 -2145.806,E2 -2145.806} C_VEL
LIN {X 0,Y 573.257,Z 308.075,A -85,B 0,C 180,E1 -2148.745,E2 -2148.745} C_VEL
LIN {X 0,Y 573.285,Z 308.078,A -85,B 0,C 180,E1 -2151.54,E2 -2151.54} C_VEL
LIN {X 0,Y 573.299,Z 308.071,A -85,B 0,C 180,E1 -2154.372,E2 -2154.372} C_VEL
LIN {X 0,Y 573.309,Z 308.07,A -85,B 0,C 180,E1 -2157.892,E2 -2157.892} C_VEL
LIN {X 0,Y 573.305,Z 308.069,A -85,B 0,C 180,E1 -2160.702,E2 -2160.702} C_VEL
LIN {X 0,Y 573.286,Z 308.072,A -85,B 0,C 180,E1 -2162.811,E2 -2162.811} C_VEL
LIN {X 0,Y 573.301,Z 308.071,A -85,B 0,C 180,E1 -2165.628,E2 -2165.628} C_VEL
LIN {X 0,Y 573.303,Z 308.075,A -85,B 0,C 180,E1 -2168.459,E2 -2168.459} C_VEL
LIN {X 0,Y 573.265,Z 308.073,A -85,B 0,C 180,E1 -2171.312,E2 -2171.312} C_VEL
LIN {X 0,Y 573.247,Z 308.076,A -85,B 0,C 180,E1 -2174.413,E2 -2174.413} C_VEL
LIN {X 0,Y 573.252,Z 308.082,A -85,B 0,C 180,E1 -2177.112,E2 -2177.112} C_VEL
LIN {X 0,Y 573.252,Z 308.077,A -85,B 0,C 180,E1 -2180.077,E2 -2180.077} C_VEL
LIN {X 0,Y 573.234,Z 308.084,A -85,B 0,C 180,E1 -2182.338,E2 -2182.338} C_VEL
LIN {X 0,Y 573.24,Z 308.08,A -85,B 0,C 180,E1 -2185.411,E2 -2185.411} C_VEL
LIN {X 0,Y 573.192,Z 308.083,A -85,B 0,C 180,E1 -2188.567,E2 -2188.567} C_VEL
LIN {X 0,Y 573.223,Z 308.085,A -85,B 0,C 180,E1 -2190.994,E2 -2190.994} C_VEL
LIN {X 0,Y 573.259,Z 308.075,A -85,B 0,C 180,E1 -2193.524,E2 -2193.524} C_VEL
LIN {X 0,Y 573.254,Z 308.081,A -85,B 0,C 180,E1 -2196.049,E2 -2196.049} C_VEL
LIN {X 0,Y 573.233,Z 308.078,A -85,B 0,C 180,E1 -2198.702,E2 -2198.702} C_VEL
LIN {X 0,Y 573.205,Z 308.083,A -85,B 0,C 180,E1 -2201.591,E2 -2201.591} C_VEL
LIN {X 0,Y 573.21,Z 308.087,A -85,B 0,C 180,E1 -2204.674,E2 -2204.674} C_VEL
LIN {X 0,Y 573.239,Z 308.08,A -85,B 0,C 180,E1 -2207.6,E2 -2207.6} C_VEL
LIN {X 0,Y 573.241,Z 308.078,A -85,B 0,C 180,E1 -2210.569,E2 -2210.569} C_VEL
LIN {X 0,Y 573.235,Z 308.109,A -85,B 0,C 180,E1 -2213.624,E2 -2213.624} C_VEL
LIN {X 0,Y 573.571,Z 311.17,A -85,B 0,C 180,E1 -2214.838,E2 -2214.838} C_VEL
LIN {X 0,Y 573.464,Z 318.838,A -85,B 0,C 180,E1 -2217.739,E2 -2217.739} C_VEL
LIN {X 0,Y 573.449,Z 326.753,A -85,B 0,C 180,E1 -2220.645,E2 -2220.645} C_VEL
LIN {X 0,Y 573.312,Z 335.657,A -85,B 0,C 180,E1 -2223.813,E2 -2223.813} C_VEL
LIN {X 0,Y 573.249,Z 343.449,A -85,B 0,C 180,E1 -2226.519,E2 -2226.519} C_VEL
LIN {X 0,Y 573.185,Z 351.239,A -85,B 0,C 180,E1 -2229.171,E2 -2229.171} C_VEL
LIN {X 0,Y 573.138,Z 359.031,A -85,B 0,C 180,E1 -2231.779,E2 -2231.779} C_VEL
LIN {X 0,Y 573.107,Z 366.822,A -85,B 0,C 180,E1 -2234.349,E2 -2234.349} C_VEL
LIN {X 0,Y 573.064,Z 375.726,A -85,B 0,C 180,E1 -2237.247,E2 -2237.247} C_VEL
LIN {X 0,Y 573.044,Z 376.491,A -85,B 0,C 180,E1 -2237.494,E2 -2237.494} C_VEL
LIN {X 0,Y 573.874,Z 382.368,A -85,B 0,C 180,E1 -2237.625,E2 -2237.625} C_VEL
LIN {X 0,Y 573.771,Z 394.494,A -85,B 0,C 180,E1 -2237.936,E2 -2237.936} C_VEL
LIN {X 0,Y 573.65,Z 406.318,A -85,B 0,C 180,E1 -2238.373,E2 -2238.373} C_VEL
LIN {X 0,Y 573.507,Z 418.492,A -85,B 0,C 180,E1 -2238.977,E2 -2238.977} C_VEL
LIN {X 0,Y 573.446,Z 429.476,A -85,B 0,C 180,E1 -2239.674,E2 -2239.674} C_VEL
LIN {X 0,Y 573.308,Z 439.645,A -85,B 0,C 180,E1 -2240.474,E2 -2240.474} C_VEL
LIN {X 0,Y 573.215,Z 448.786,A -85,B 0,C 180,E1 -2241.362,E2 -2241.362} C_VEL
LIN {X 0,Y 573.142,Z 457.689,A -85,B 0,C 180,E1 -2242.425,E2 -2242.425} C_VEL
LIN {X 0,Y 573.051,Z 464.405,A -85,B 0,C 180,E1 -2243.415,E2 -2243.415} C_VEL
LIN {X 0,Y 573.07,Z 469.679,A -85,B 0,C 180,E1 -2244.369,E2 -2244.369} C_VEL
LIN {X 0,Y 573.028,Z 474.371,A -85,B 0,C 180,E1 -2245.427,E2 -2245.427} C_VEL
LIN {X 0,Y 573.022,Z 477.956,A -85,B 0,C 180,E1 -2246.484,E2 -2246.484} C_VEL
LIN {X 0,Y 572.959,Z 479.808,A -85,B 0,C 180,E1 -2247.187,E2 -2247.187} C_VEL
LIN {X 0,Y 572.94,Z 481.2,A -85,B 0,C 180,E1 -2247.891,E2 -2247.891} C_VEL
LIN {X 0,Y 572.94,Z 482.784,A -85,B 0,C 180,E1 -2249.297,E2 -2249.297} C_VEL
LIN {X 0,Y 572.938,Z 483,A -85,B 0,C 180,E1 -2250,E2 -2250} C_VEL
LIN {X 0,Y 572.946,Z 482.185,A -85,B 0,C 180,E1 -2251.405,E2 -2251.405} C_VEL
LIN {X 0,Y 572.94,Z 481.202,A -85,B 0,C 180,E1 -2252.109,E2 -2252.109} C_VEL
LIN {X 0,Y 572.959,Z 479.81,A -85,B 0,C 180,E1 -2252.812,E2 -2252.812} C_VEL
LIN {X 0,Y 573.014,Z 476.897,A -85,B 0,C 180,E1 -2253.868,E2 -2253.868} C_VEL
LIN {X 0,Y 572.963,Z 472.951,A -85,B 0,C 180,E1 -2254.925,E2 -2254.925} C_VEL
LIN {X 0,Y 573.065,Z 466.88,A -85,B 0,C 180,E1 -2256.16,E2 -2256.16} C_VEL
LIN {X 0,Y 573.119,Z 460.239,A -85,B 0,C 180,E1 -2257.22,E2 -2257.22} C_VEL
LIN {X 0,Y 573.2,Z 451.994,A -85,B 0,C 180,E1 -2258.283,E2 -2258.283} C_VEL
LIN {X 0,Y 573.286,Z 443.543,A -85,B 0,C 180,E1 -2259.17,E2 -2259.17} C_VEL
LIN {X 0,Y 573.425,Z 433.101,A -85,B 0,C 180,E1 -2260.058,E2 -2260.058} C_VEL
LIN {X 0,Y 573.511,Z 421.545,A -85,B 0,C 180,E1 -2260.847,E2 -2260.847} C_VEL
LIN {X 0,Y 573.61,Z 409.891,A -85,B 0,C 180,E1 -2261.466,E2 -2261.466} C_VEL
LIN {X 0,Y 573.763,Z 397.191,A -85,B 0,C 180,E1 -2261.973,E2 -2261.973} C_VEL
LIN {X 0,Y 573.854,Z 384.545,A -85,B 0,C 180,E1 -2262.33,E2 -2262.33} C_VEL
LIN {X 0,Y 573.674,Z 380.681,A -85,B 0,C 180,E1 -2262.413,E2 -2262.413} C_VEL
LIN {X 0,Y 573.043,Z 376.493,A -85,B 0,C 180,E1 -2262.505,E2 -2262.505} C_VEL
LIN {X 0,Y 573.084,Z 367.937,A -85,B 0,C 180,E1 -2265.287,E2 -2265.287} C_VEL
LIN {X 0,Y 573.146,Z 360.146,A -85,B 0,C 180,E1 -2267.851,E2 -2267.851} C_VEL
LIN {X 0,Y 573.198,Z 352.354,A -85,B 0,C 180,E1 -2270.452,E2 -2270.452} C_VEL
LIN {X 0,Y 573.221,Z 344.443,A -85,B 0,C 180,E1 -2273.141,E2 -2273.141} C_VEL
LIN {X 0,Y 573.287,Z 336.772,A -85,B 0,C 180,E1 -2275.797,E2 -2275.797} C_VEL
LIN {X 0,Y 573.349,Z 328.981,A -85,B 0,C 180,E1 -2278.557,E2 -2278.557} C_VEL
LIN {X 0,Y 573.428,Z 322.302,A -85,B 0,C 180,E1 -2280.98,E2 -2280.98} C_VEL
LIN {X 0,Y 573.525,Z 315.363,A -85,B 0,C 180,E1 -2283.563,E2 -2283.563} C_VEL
LIN {X 0,Y 573.538,Z 310.1,A -85,B 0,C 180,E1 -2285.578,E2 -2285.578} C_VEL
LIN {X 0,Y 573.24,Z 308.084,A -85,B 0,C 180,E1 -2286.429,E2 -2286.429} C_VEL
LIN {X 0,Y 573.247,Z 308.077,A -85,B 0,C 180,E1 -2289.432,E2 -2289.432} C_VEL
LIN {X 0,Y 573.25,Z 308.079,A -85,B 0,C 180,E1 -2291.595,E2 -2291.595} C_VEL
LIN {X 0,Y 573.234,Z 308.079,A -85,B 0,C 180,E1 -2294.332,E2 -2294.332} C_VEL
LIN {X 0,Y 573.216,Z 308.084,A -85,B 0,C 180,E1 -2297.36,E2 -2297.36} C_VEL
LIN {X 0,Y 573.233,Z 308.082,A -85,B 0,C 180,E1 -2300.392,E2 -2300.392} C_VEL
